// TIA Portal V18 program export: 1 tag tables, 60 data types, 57 data blocks, 79 code blocks (in call order from the OBs), 25 instance data blocks

VAR_GLOBAL   // PLC tag table "Default tag table"
   "AI11.02.01" AT %IW96 : Int;
   "AI12.01.01" AT %IW68 : Int;
   "AI12.01.02" AT %IW70 : Int;
   "AI12.01.03" AT %IW72 : Int;
   "AI12.01.04" AT %IW74 : Int;
   "AI12.01.05" AT %IW76 : Int;
   "AI12.01.06" AT %IW78 : Int;
   "AI12.01.07" AT %IW80 : Int;
   "AI12.01.08" AT %IW82 : Int;
   "AI11.02.02" AT %IW98 : Int;
   "AI11.02.03" AT %IW100 : Int;
   "AI11.02.04" AT %IW102 : Int;
   "AI11.02.05" AT %IW104 : Int;
   "AI11.02.06" AT %IW106 : Int;
   "AI11.02.07" AT %IW108 : Int;
   "AI11.02.08" AT %IW110 : Int;
   "AI11.03.01" AT %IW112 : Int;
   "AI11.03.02" AT %IW114 : Int;
   "AI11.03.03" AT %IW116 : Int;
   "AI11.03.04" AT %IW118 : Int;
   "AI11.03.05" AT %IW120 : Int;
   "AI11.03.06" AT %IW122 : Int;
   "AI11.03.07" AT %IW124 : Int;
   "AI11.03.08" AT %IW126 : Int;
   "AO12.02.01" AT %QW68 : Int;
   "AO12.02.02" AT %QW70 : Int;
   "AO12.02.03" AT %QW72 : Int;
   "AO12.02.04" AT %QW74 : Int;
   "AO12.02.05" AT %QW76 : Int;
   "AO12.02.06" AT %QW78 : Int;
   "AO12.02.07" AT %QW80 : Int;
   "AO12.02.08" AT %QW82 : Int;
   "DI12.03.01" AT %I2.0 : Bool;
   "DI12.03.02" AT %I2.1 : Bool;
   "DI12.03.03" AT %I2.2 : Bool;
   "DI12.03.04" AT %I2.3 : Bool;
   "DI12.03.05" AT %I2.4 : Bool;
   "DI12.03.06" AT %I2.5 : Bool;
   "DI12.03.07" AT %I2.6 : Bool;
   "DI12.03.08" AT %I2.7 : Bool;
   "DI12.03.09" AT %I3.0 : Bool;
   "DI12.03.10" AT %I3.1 : Bool;
   "DI12.03.11" AT %I3.2 : Bool;
   "DI12.03.12" AT %I3.3 : Bool;
   "DI12.03.13" AT %I3.4 : Bool;
   "DI12.03.14" AT %I3.5 : Bool;
   "DI12.03.15" AT %I3.6 : Bool;
   "DI12.03.16" AT %I3.7 : Bool;
   "DI12.03.17" AT %I4.0 : Bool;
   "DI12.03.18" AT %I4.1 : Bool;
   "DI12.03.19" AT %I4.2 : Bool;
   "DI12.03.20" AT %I4.3 : Bool;
   "DI12.03.21" AT %I4.4 : Bool;
   "DI12.03.22" AT %I4.5 : Bool;
   "DI12.03.23" AT %I4.6 : Bool;
   "DI12.03.24" AT %I4.7 : Bool;
   "DI12.03.25" AT %I5.0 : Bool;
   "DI12.03.26" AT %I5.1 : Bool;
   "DI12.03.27" AT %I5.2 : Bool;
   "DI12.03.28" AT %I5.3 : Bool;
   "DI12.03.29" AT %I5.4 : Bool;
   "DI12.03.30" AT %I5.5 : Bool;
   "DI12.03.31" AT %I5.6 : Bool;
   "DI12.03.32" AT %I5.7 : Bool;
   "DO12.04.01" AT %Q2.0 : Bool;
   "DO12.04.02" AT %Q2.1 : Bool;
   "DO12.04.03" AT %Q2.2 : Bool;
   "DO12.04.04" AT %Q2.3 : Bool;
   "DO12.04.05" AT %Q2.4 : Bool;
   "DO12.04.06" AT %Q2.5 : Bool;
   "DO12.04.07" AT %Q2.6 : Bool;
   "DO12.04.08" AT %Q2.7 : Bool;
   "DO12.04.09" AT %Q3.0 : Bool;
   "DO12.04.10" AT %Q3.1 : Bool;
   "DO12.04.11" AT %Q3.2 : Bool;
   "DO12.04.12" AT %Q3.3 : Bool;
   "DO12.04.13" AT %Q3.4 : Bool;
   "DO12.04.14" AT %Q3.5 : Bool;
   "DO12.04.15" AT %Q3.6 : Bool;
   "DO12.04.16" AT %Q3.7 : Bool;
   "DO12.04.17" AT %Q4.0 : Bool;
   "DO12.04.18" AT %Q4.1 : Bool;
   "DO12.04.19" AT %Q4.2 : Bool;
   "DO12.04.20" AT %Q4.3 : Bool;
   "DO12.04.21" AT %Q4.4 : Bool;
   "DO12.04.22" AT %Q4.5 : Bool;
   "DO12.04.23" AT %Q4.6 : Bool;
   "DO12.04.24" AT %Q4.7 : Bool;
   "DO12.04.25" AT %Q5.0 : Bool;
   "DO12.04.26" AT %Q5.1 : Bool;
   "DO12.04.27" AT %Q5.2 : Bool;
   "DO12.04.28" AT %Q5.3 : Bool;
   "DO12.04.29" AT %Q5.4 : Bool;
   "DO12.04.30" AT %Q5.5 : Bool;
   "DO12.04.31" AT %Q5.6 : Bool;
   "DO12.04.32" AT %Q5.7 : Bool;
   "DI11.05.01" AT %I16.0 : Bool;
   "DI11.05.02" AT %I16.1 : Bool;
   "DI11.05.03" AT %I16.2 : Bool;
   "DI11.05.04" AT %I16.3 : Bool;
   "DI11.05.05" AT %I16.4 : Bool;
   "DI11.05.06" AT %I16.5 : Bool;
   "DI11.05.07" AT %I16.6 : Bool;
   "DI11.05.08" AT %I16.7 : Bool;
   "DI11.05.09" AT %I17.0 : Bool;
   "DI11.05.10" AT %I17.1 : Bool;
   "DI11.05.11" AT %I17.2 : Bool;
   "DI11.05.12" AT %I17.3 : Bool;
   "DI11.05.13" AT %I17.4 : Bool;
   "DI11.05.14" AT %I17.5 : Bool;
   "DI11.05.15" AT %I17.6 : Bool;
   "DI11.05.16" AT %I17.7 : Bool;
   "DI11.06.01" AT %I20.0 : Bool;
   "DI11.06.02" AT %I20.1 : Bool;
   "DI11.06.03" AT %I20.2 : Bool;
   "DI11.06.04" AT %I20.3 : Bool;
   "DI11.06.05" AT %I20.4 : Bool;
   "DI11.06.06" AT %I20.5 : Bool;
   "DI11.06.07" AT %I20.6 : Bool;
   "DI11.06.08" AT %I20.7 : Bool;
   "DI11.06.09" AT %I21.0 : Bool;
   "DI11.06.10" AT %I21.1 : Bool;
   "DI11.06.11" AT %I21.2 : Bool;
   "DI11.06.12" AT %I21.3 : Bool;
   "DI11.06.13" AT %I21.4 : Bool;
   "DI11.06.14" AT %I21.5 : Bool;
   "DI11.06.15" AT %I21.6 : Bool;
   "DI11.06.16" AT %I21.7 : Bool;
   "DI11.07.01" AT %I28.0 : Bool;
   "DI11.07.02" AT %I28.1 : Bool;
   "DI11.07.03" AT %I28.2 : Bool;
   "DI11.07.04" AT %I28.3 : Bool;
   "DI11.07.05" AT %I28.4 : Bool;
   "DI11.07.06" AT %I28.5 : Bool;
   "DI11.07.07" AT %I28.6 : Bool;
   "DI11.07.08" AT %I28.7 : Bool;
   "DI11.07.09" AT %I29.0 : Bool;
   "DI11.07.10" AT %I29.1 : Bool;
   "DI11.07.11" AT %I29.2 : Bool;
   "DI11.07.12" AT %I29.3 : Bool;
   "DI11.07.13" AT %I29.4 : Bool;
   "DI11.07.14" AT %I29.5 : Bool;
   "DI11.07.15" AT %I29.6 : Bool;
   "DI11.07.16" AT %I29.7 : Bool;
   "DO11.07.01" AT %Q28.0 : Bool;
   "DO11.07.02" AT %Q28.1 : Bool;
   "DO11.07.03" AT %Q28.2 : Bool;
   "DO11.07.04" AT %Q28.3 : Bool;
   "DO11.07.05" AT %Q28.4 : Bool;
   "DO11.07.06" AT %Q28.5 : Bool;
   "DO11.07.07" AT %Q28.6 : Bool;
   "DO11.07.08" AT %Q28.7 : Bool;
   "DO11.07.09" AT %Q29.0 : Bool;
   "DO11.07.10" AT %Q29.1 : Bool;
   "DI11.08.01" AT %I32.0 : Bool;
   "DI11.08.02" AT %I32.1 : Bool;
   "DI11.08.03" AT %I32.2 : Bool;
   "DI11.08.04" AT %I32.3 : Bool;
   "DI11.08.05" AT %I32.4 : Bool;
   "DI11.08.06" AT %I32.5 : Bool;
   "DI11.08.07" AT %I32.6 : Bool;
   "DI11.08.08" AT %I32.7 : Bool;
   "DI11.08.09" AT %I33.0 : Bool;
   "DI11.08.10" AT %I33.1 : Bool;
   "DI11.08.11" AT %I33.2 : Bool;
   "DI11.08.12" AT %I33.3 : Bool;
   "DI11.08.13" AT %I33.4 : Bool;
   "DI11.08.14" AT %I33.5 : Bool;
   "DI11.08.15" AT %I33.6 : Bool;
   "DI11.08.16" AT %I33.7 : Bool;
   "DI11.01.01" AT %I0.0 : Bool;
   "DI11.01.02" AT %I0.1 : Bool;
   "DI11.01.03" AT %I0.2 : Bool;
   "DI11.01.04" AT %I0.3 : Bool;
   "DI11.01.05" AT %I0.4 : Bool;
   "DI11.01.06" AT %I0.5 : Bool;
   "DI11.01.07" AT %I0.6 : Bool;
   "DI11.01.08" AT %I0.7 : Bool;
   "DI11.01.09" AT %I1.0 : Bool;
   "DI11.01.10" AT %I1.1 : Bool;
   "DI11.01.11" AT %I1.2 : Bool;
   "DI11.01.12" AT %I1.3 : Bool;
   "DI11.01.13" AT %I1.4 : Bool;
   "DI11.01.14" AT %I1.5 : Bool;
   "DO11.07.11" AT %Q29.2 : Bool;
   "DO11.07.12" AT %Q29.3 : Bool;
   "DO11.07.13" AT %Q29.4 : Bool;
   "DO11.07.14" AT %Q29.5 : Bool;
   "DO11.07.15" AT %Q29.6 : Bool;
   "DO11.07.16" AT %Q29.7 : Bool;
   "DO11.08.01" AT %Q32.0 : Bool;
   "DO11.08.02" AT %Q32.1 : Bool;
   "DO11.08.03" AT %Q32.2 : Bool;
   "DO11.08.04" AT %Q32.3 : Bool;
   "DO11.08.05" AT %Q32.4 : Bool;
   "DO11.08.06" AT %Q32.5 : Bool;
   "DO11.08.07" AT %Q32.6 : Bool;
   "DO11.08.08" AT %Q32.7 : Bool;
   "DO11.08.09" AT %Q33.0 : Bool;
   "DO11.08.10" AT %Q33.1 : Bool;
   "DO11.08.11" AT %Q33.2 : Bool;
   "DO11.08.12" AT %Q33.3 : Bool;
   "DO11.08.13" AT %Q33.4 : Bool;
   "DO11.08.14" AT %Q33.5 : Bool;
   "DO11.08.15" AT %Q33.6 : Bool;
   "DO11.08.16" AT %Q33.7 : Bool;
   "AO11.04.01" AT %QW128 : Int;
   "AO11.04.02" AT %QW130 : Int;
   "AO11.04.03" AT %QW132 : Int;
   "AO11.04.04" AT %QW134 : Int;
   "DO11.01.01" AT %Q0.0 : Bool;
   "DO11.01.02" AT %Q0.1 : Bool;
   "DO11.01.03" AT %Q0.2 : Bool;
   "DO11.01.04" AT %Q0.3 : Bool;
   "DO11.01.05" AT %Q0.4 : Bool;
   "DO11.01.06" AT %Q0.5 : Bool;
   "DO11.01.07" AT %Q0.6 : Bool;
   "DO11.01.08" AT %Q0.7 : Bool;
   "DO11.01.09" AT %Q1.0 : Bool;
   "DO11.01.10" AT %Q1.1 : Bool;
   "AI11.01.01" AT %IW64 : Int;
   "AI11.01.02" AT %IW66 : Int;
   "AO11.01.01" AT %QW64 : Int;
   "AO11.01.02" AT %QW66 : Int;
   System_Byte AT %MB1 : Byte;
   FirstScan AT %M1.0 : Bool;
   DiagStatusUpdate AT %M1.1 : Bool;
   AlwaysTRUE AT %M1.2 : Bool;
   AlwaysFALSE AT %M1.3 : Bool;
   Clock_Byte AT %MB0 : Byte;
   Clock_10Hz AT %M0.0 : Bool;
   Clock_5Hz AT %M0.1 : Bool;
   "Clock_2.5Hz" AT %M0.2 : Bool;
   Clock_2Hz AT %M0.3 : Bool;
   "Clock_1.25Hz" AT %M0.4 : Bool;
   Clock_1Hz AT %M0.5 : Bool;
   "Clock_0.625Hz" AT %M0.6 : Bool;
   "Clock_0.5Hz" AT %M0.7 : Bool;
   Lux AT %MD20 : Real;
   "DI12.05.01" AT %I6.0 : Bool;
   "DI12.05.02" AT %I6.1 : Bool;
   "DI12.05.03" AT %I6.2 : Bool;
   "DI12.05.04" AT %I6.3 : Bool;
   "DI12.05.05" AT %I6.4 : Bool;
   "DI12.05.06" AT %I6.5 : Bool;
   "DI12.05.07" AT %I6.6 : Bool;
   "DI12.05.08" AT %I6.7 : Bool;
   "DI12.05.09" AT %I7.0 : Bool;
   "DI12.05.10" AT %I7.1 : Bool;
   "DI12.05.11" AT %I7.2 : Bool;
   "DI12.05.12" AT %I7.3 : Bool;
   "DI12.05.13" AT %I7.4 : Bool;
   "DI12.05.14" AT %I7.5 : Bool;
   "DI12.05.15" AT %I7.6 : Bool;
   "DI12.05.16" AT %I7.7 : Bool;
   OAT_clock_triger AT %M5.0 : Bool;
   "Run/Stop" AT %M5.1 : Bool;
   rAO_temporary AT %MD60 : Real;
   rAI_temporary AT %MD61 : Real;
   xDO_temporary AT %M5.2 : Bool;   //    {ExternalWritable false}
   xDI_temporary AT %M5.3 : Bool;
   iUnitStateCounter AT %MW66 : Int;
   iTargetUnitStareCounter AT %MW68 : Int;
   cTargetUnitStatePrevOne AT %MB8 : Byte;
   cActualOpModePrevOne AT %MB9 : Byte;
   iActualOpModeCounter AT %MW10 : Int;
   xDL_Pump1_Run AT %M12.0 : Bool;
   xDL_Pump2_Run AT %M12.1 : Bool;
END_VAR
VAR_GLOBAL CONSTANT   // user constants
   IOmark_string_length : Int := 25;
   DIbasic_OnDelayCycle : Int := 800;
   DIbasic_OffDelayCycle : Int := 800;
END_VAR

TYPE "UDT_DailyScheduler"
// stored: IsFailsafeCompliant false
   STRUCT
      Start : Time_Of_Day;
      Stop : Time_Of_Day;
   END_STRUCT;
END_TYPE

TYPE "UDT_Store_OpMode"
// stored: IsFailsafeCompliant false
   STRUCT
      cPreviousOne { S7_SetPoint := 'True'} : Byte;
      cActual { S7_SetPoint := 'True'} : Byte;   // Поточний/Актуальний режим роботи
      cTarget { S7_SetPoint := 'True'} : Byte;   // Вибраний режим роботи, але ще не дійшли до нього
      cPreselectedOpMode : Byte;   // 0-Protection/1-economy/2-PreComfort/3-Comfort/4-Auto
   END_STRUCT;
END_TYPE

TYPE "UDT_Store_Setpoints"
// stored: IsFailsafeCompliant false
   STRUCT
      Room : Struct
         Actual : Struct
            rRATHeating : Real;
            rRATCooling : Real;
            rIAQ : Real;
            rBuildingdP : Real;
         END_STRUCT;
         Comfort : Struct
            rRATHeating : Real := 18.0;
            rRATCooling : Real := 22.0;
            rIAQ : Real := 600.0;
            rBuildingdP : Real := 5.0;
         END_STRUCT;
         PreComfort : Struct
            rRATHeating : Real := 16.0;
            rRATCooling : Real := 25.0;
            rIAQ : Real := 800.0;
            rBuildingdP : Real := 2.0;
         END_STRUCT;
         Econom : Struct
            rRATHeating : Real := 15.0;
            rRATCooling : Real := 30.0;
            rIAQ : Real;
            rBuildingdP : Real;
         END_STRUCT;
         Protection : Struct
            rRATHeating : Real := 5.0;
            rRATCooling : Real := 35.0;
            rIAQ : Real := 0.0;
            rBuildingdP : Real := 0.0;
         END_STRUCT;
      END_STRUCT;
   END_STRUCT;
END_TYPE

TYPE "UDT_WeatherCompCurve"
// stored: IsFailsafeCompliant false
   STRUCT
      rEffectiveRoomSetPoint : Array[0..2] of Real;
      rHeatingCurveLevel : Array[0..2] of Real;
      rHeatingCurveSlope : Array[0..2] of Real;
      rSetpointTemp : Array[0..2] of Real;
      rOATforHeatingCurves : Array[0..2] of Real;
   END_STRUCT;
   // rEffectiveRoomSetPoint[0] := 20.0;
   // rEffectiveRoomSetPoint[1] := 21.0;
   // rEffectiveRoomSetPoint[2] := 22.0;
   // rHeatingCurveLevel[1] := 1.0;
   // rHeatingCurveLevel[2] := 2.0;
   // rHeatingCurveSlope[0] := 2.0;
   // rHeatingCurveSlope[1] := 2.1;
   // rHeatingCurveSlope[2] := 2.2;
   // rSetpointTemp[0] := 50.0;
   // rSetpointTemp[1] := 51.0;
   // rSetpointTemp[2] := 52.0;
END_TYPE

TYPE "UDT_OAT"
// stored: IsFailsafeCompliant false
   STRUCT
      rOAT_PLC_IO : Real;
      rOAT_WeatherStation : Real;
      rOAT_Boilers : Real;
      rOAT_Actual : Real;
   END_STRUCT;
END_TYPE

TYPE "UDT_Store_Holidays"
// stored: IsFailsafeCompliant false
   STRUCT
      UDT_Store_Holidays : Array[0..7] of Date;
   END_STRUCT;
END_TYPE

TYPE "UDT_Store_Scheduler"
// stored: IsFailsafeCompliant false
   STRUCT
      cOpModeNowByScheduler : Byte;
      Monday : Struct
         Comfort { S7_SetPoint := 'True'} : "UDT_DailyScheduler";
         PreComfort { S7_SetPoint := 'True'} : "UDT_DailyScheduler";
      END_STRUCT;
      WorkingDays : Struct
         Comfort { S7_SetPoint := 'True'} : "UDT_DailyScheduler";
         PreComfort { S7_SetPoint := 'True'} : "UDT_DailyScheduler";
      END_STRUCT;
      Saturday : Struct
         Comfort { S7_SetPoint := 'True'} : "UDT_DailyScheduler";
         PreComfort { S7_SetPoint := 'True'} : "UDT_DailyScheduler";
      END_STRUCT;
      Sunday : Struct
         Comfort { S7_SetPoint := 'True'} : "UDT_DailyScheduler";
         PreComfort { S7_SetPoint := 'True'} : "UDT_DailyScheduler";
      END_STRUCT;
      Holiday : Struct
         Comfort { S7_SetPoint := 'True'} : "UDT_DailyScheduler";
         PreComfort { S7_SetPoint := 'True'} : "UDT_DailyScheduler";
      END_STRUCT;
   END_STRUCT;
END_TYPE

TYPE "UDT_Store_Season"
// stored: IsFailsafeCompliant false
   STRUCT
      cSeasonModeSelection : Byte;   // 0 = Summer 1 = Winter 2 = Midseason, 3=Auro
      cActual : Byte;   // 0 = Summer 1 = Winter 2 = Midseason
      cTarget : Byte;
      cReserve : Byte;
      rOATtoWinter : Real := 10.0;
      rOATtoSummer : Real := 12.0;
   END_STRUCT;
END_TYPE

TYPE "UDT_DL_Vars"
// stored: IsFailsafeCompliant false
   STRUCT
      rOATtoHeatUpLine : Real;
      cReserve1 : Byte;
      cReserve2 : Byte;
      cDLPanelModeSelector : Byte := 16#3;
      rDayTankLevelAlarmMin : Array[1..2] of Real;
      rDayTankLevelStartFilling : Array[1..2] of Real;
      rDayTankLevelStopFilling : Array[1..2] of Real;
      rDayTankLevelAlarmMax : Array[1..2] of Real;
      cExericeSeconds : Array[1..2] of Byte;
      cMaxHoursWithoutRunToExerise : Array[1..2] of Byte;
      cActualHoursWithoutRunToExerise : Array[1..2] of Byte;
   END_STRUCT;
   // rDayTankLevelAlarmMin[1] := 50.0;
   // rDayTankLevelAlarmMin[2] := 51.0;
   // rDayTankLevelStartFilling[1] := 70.0;
   // rDayTankLevelStartFilling[2] := 71.0;
   // rDayTankLevelStopFilling[1] := 90.0;
   // rDayTankLevelStopFilling[2] := 91.1;
   // rDayTankLevelAlarmMax[1] := 95.0;
   // rDayTankLevelAlarmMax[2] := 96.0;
   // cExericeSeconds[1..2] := 16#FA;
   // cMaxHoursWithoutRunToExerise[1] := 16#A8;
   // cMaxHoursWithoutRunToExerise[2] := 16#A9;
END_TYPE

TYPE "UDT_BoilersOnOffSettings"
// stored: IsFailsafeCompliant false
   STRUCT
      OAT : Struct
         rBoiler1OATOff : Real := 18.0;
         rBoiler1OATOn : Real := 15.0;
         rBoiler2OAT1On : Real := 5.0;
         rBoiler2OAT1Off : Real := 10.0;
         rBoiler2OAT2On : Real := -5.0;
         rBoiler2OAT2Off : Real;
      END_STRUCT;
      PLCModeSelection : Struct
         cPreselectedOpModePLC : Byte;   // Вибор режиму роботи з PLC. 0-Вимкенено/1-Boiler1/2-Boiler2/3-B1+B2/4-Auto
         cActualOpModePLC : Byte;   // Актуальний режим роботи з PLC. 0-Вимкенено/1-Boiler1/2-Boiler2/3-B1+B2/4-Auto
      END_STRUCT;
   END_STRUCT;
END_TYPE

TYPE "UDT_Vitotronic100_Alarms"
// stored: IsFailsafeCompliant false
   STRUCT
      "00 General alarm" : Array[0..2] of Bool;
   END_STRUCT;
END_TYPE

TYPE "UDT_Vitotronic100_IOs"
// stored: IsFailsafeCompliant false
   STRUCT
      "Boiler water temperature" : Array[0..2] of Real;
      "Flue gas temperature" : Array[0..2] of Real;
      "Return temperature 17A" : Array[0..2] of Real;
      "Return temperature 17B" : Array[0..2] of Real;
   END_STRUCT;
END_TYPE

TYPE "UDT_Vitotronic100_Params"
// stored: IsFailsafeCompliant false
   STRUCT
      "Actual system output - value" : Array[0..2] of Real;
      "Boiler output value" : Array[0..2] of Real;
      "Burner output" : Array[0..2] of Real;
      "Maximum boiler temperature" : Array[0..2] of Real;
      "Minimum boiler temperature" : Array[0..2] of Real;
      "Set boiler output (effective)" : Array[0..2] of Real;
      "Set boiler water temperature (effective)" : Array[0..2] of Real;
   END_STRUCT;
END_TYPE

TYPE "UDT_BoilersSummaryAlarms"
// stored: IsFailsafeCompliant false
   STRUCT
      BlockingAlarm : Array[1..2] of Bool;
   END_STRUCT;
END_TYPE

TYPE "UDT_Vitotronic100_Settings"
// stored: IsFailsafeCompliant false
   STRUCT
      "Set boiler water temperature" : Array[0..2] of Real;
      "Operating mode system_boiler" : Array[0..2] of Int;
   END_STRUCT;
END_TYPE

TYPE "UDT_BoilerOpMode"
// stored: IsFailsafeCompliant false
   STRUCT
      cPreviousOne { S7_SetPoint := 'True'} : Array[1..2] of Byte;
      cActual { S7_SetPoint := 'True'} : Array[1..2] of Byte;   // Поточний/Актуальний режим роботи
      cTarget { S7_SetPoint := 'True'} : Array[1..2] of Byte;   // Вибраний режим роботи, але ще не дійшли до нього
      cPreselectedOpModePLC : Array[1..2] of Byte;   // Вибор режиму роботи з PLC. 0-Вимкенено/1-Boiler1/2-Boiler2/3-B1+B2/4-Auto
      cReserve : Array[1..2] of Byte;
      cPreselectedOpModePanel : Array[1..2] of Byte;   // Вибор режиму роботи з Фізичного перемикача на шафы. 0-Summer/1-Winter/2--Auto
      xBoiler2IndividualPanelSwitch : Bool;
   END_STRUCT;
END_TYPE

TYPE "UDT_BoilerUnitState"
// stored: IsFailsafeCompliant false
   STRUCT
      iBoilerSimpleState : Array[1..2] of Int;   // 0-Off, 1 - Heating, 2 - Alarm
      xBoilerOATRequest : Array[1..2] of Bool;
      xBoilerRequestedByAlarm : Array[1..2] of Bool;
      cTarget : Array[1..2] of Byte;
      cActual : Array[1..2] of Byte;
   END_STRUCT;
END_TYPE

TYPE "UDT_AIbasic"
// stored: IsFailsafeCompliant false
   STRUCT
      iID : DInt;   // AIs ID for monitoring
      iValue : Int;   // Int value
      rValue : Real;   // Real value
      iFilterSet : Int;   // Filter value
      rMin : Real;   // Scale Min
      rMax : Real;   // Scale Max
      wMark : String["IOmark_string_length"];   // AIs label for monitoring
   END_STRUCT;
END_TYPE

TYPE "UDT_AObasic"
// stored: IsFailsafeCompliant false
   STRUCT
      iID : DInt;   // AOs ID for monitoring
      rInput : Real;   // Value for AO
      cMOA : Byte;   // Mode Manual/Off/Auto
      rMan_output : Real;   // Manual output
      iOutput : Int;   // Output for DAC
      wMark : String["IOmark_string_length"];   // AOs label for monitoring
   END_STRUCT;
END_TYPE

TYPE "UDT_DIbasic"
// stored: IsFailsafeCompliant false
   STRUCT
      iID : DInt;   // DIs ID for monitoring
      iCounter : Int;   // Counter for DIs EDGE
      xFiltered : Bool;   // Filtered value
      wMark : String["IOmark_string_length"];   // DIs label for monitoring
      iAddImpOff : Int;   // Temp
      iAddImpOn : Int;   // Temp
      xMemory : Bool;   // Temp
   END_STRUCT;
END_TYPE

TYPE "UDT_DObasic"
// stored: IsFailsafeCompliant false
   STRUCT
      iID : DInt;   // DOs ID for monitoring
      xInput : Bool;   // Value for DO
      cMOA : Byte;   // Mode Manual/Off/Auto
      xOutput : Bool;   // Phisicl output
      iCounter : Int;   // Counter
      Mark : String["IOmark_string_length"];   // DOs label for monitoring
      xBitCount : Bool;   // Internal
   END_STRUCT;
END_TYPE

TYPE "UDT_RTDbasic"
// stored: IsFailsafeCompliant false
   STRUCT
      iID : DInt;   // AIs ID for monitoring
      rValue : Real;   // Real value
      iFilterSet : Int;   // Filter value
      rCalibration : Real;   // Scale Min
      rDiv : Real := 100.0;   // Scale Max
      wMark : String["IOmark_string_length"];   // AIs label for monitoring
   END_STRUCT;
END_TYPE

TYPE "UDT_DLsAI"
// stored: IsFailsafeCompliant false
   STRUCT
      rDayTankLevel : Array[1..2] of Real;   // 10.82(3) Рівень палива в баку добового запасу ДГУ1(2)
   END_STRUCT;
END_TYPE

TYPE "UDT_DLsDI"
// stored: IsFailsafeCompliant false
   STRUCT
      xDieselLineHeatingReady : Array[1..2] of Bool;
      xDieselLineHeatingInd : Array[1..2] of Bool;
      xDieselLinePumpInd : Array[1..2] of Bool;
      xDieselLinePnom : Bool;   // 10.67 Номінальний тиск в ДП ліній
      xDieselLineValveToBoilerInd : Bool;   // 10.66 Клапанна група на Котел
      xDieselLinePmax : Bool;   // 10.68 Високий тиск в ДП ліній
      xDieselLinePumpZoneWaterFloodAlarm : Bool;   // 10.79 Затоплення приямку з насосами
      xDieselLineMainTankDoubleWallAlarmInd : Bool;   // 10.63 62 SGB DL-4000
      xDieselLineMainTankMinLevelInd : Bool;   // 10.75 76
      Reserve1 : Bool;
      Reserve2 : Bool;
      xDieselLinePumpPanelSelectorOff : Bool;
      xDieselLinePumpPanelSelectorP1Man : Bool;
      xDieselLinePumpPanelSelectorP2Man : Bool;
      xDieselLinePumpPanelSelectorAuto : Bool;
   END_STRUCT;
END_TYPE

TYPE "UDT_DLsDO"
// stored: IsFailsafeCompliant false
   STRUCT
      xDieselLineHeatingCmd : Array[1..2] of Bool;
      xDieselLinePumpEnable : Bool;
      xDieselLinePumpSelect : Bool;
      xDieselLineDayTankValve : Array[1..2] of Bool;
      Reserve : Array[1..2] of Bool;
   END_STRUCT;
END_TYPE

TYPE "AHUChannel_v1"
// stored: IsFailsafeCompliant false
   STRUCT
      SAFCmd1 : Array[0..2] of Bool;
      SAFCmd2 : Array[0..2] of Bool;
      SAFCmd3 : Array[0..2] of Bool;
      SAFSpeed1Ind : Array[0..2] of Bool;   // Off/On
      SAFSpeed2Ind : Array[0..2] of Bool;   // Off/On
      SAFIsBlockedByFrostProt : Array[0..2] of Bool;   // Off/On
      SAFInd4 : Array[0..2] of Bool;
      SAFInd5 : Array[0..2] of Bool;
      SAFInd6 : Array[0..2] of Bool;
      SAFInd7 : Array[0..2] of Bool;
      HeaterRlyIsOn : Array[0..2] of Bool;   // Off/On
      HeaterRlyIsOff : Array[0..2] of Bool;   // Off/On
      HeaterRlyOnCmd : Array[0..2] of Bool;   // Off/On
      HeaterInitialSignal : Array[0..2] of Real;   // 0-100.0%
      HeaterAdaptedSignal : Array[0..2] of Real;   // 0-100.0%
      MixingRlyIsOn : Array[0..2] of Bool;   // Off/On
      MixingRlyIsOff : Array[0..2] of Bool;   // Off/On
      MixingRlyOnCmd : Array[0..2] of Bool;   // Off/On
      MixingInitialSignal : Array[0..2] of Real;   // 0-100.0%
      MixingAdaptedSignal : Array[0..2] of Real;   // 0-100.0%
      ExtractRlyIsOn : Array[0..2] of Bool;   // Off/On
      ExtractRlyIsOff : Array[0..2] of Bool;   // Off/On
      ExtractRlyOnCmd : Array[0..2] of Bool;   // Off/On
      ExtractInitialSignal : Array[0..2] of Real;   // 0-100.0%
      ExtractAdaptedSignal : Array[0..2] of Real;   // 0-100.0%
   END_STRUCT;
END_TYPE

TYPE "SupplyFanChannel_v1"
// stored: IsFailsafeCompliant false
   STRUCT
      SAFSpeed1Ind : Array[0..2] of Bool;   // Off/On
      SAFSpeed2Ind : Array[0..2] of Bool;   // Off/On
      SAFIsBlockedByFrostProt : Array[0..2] of Bool;   // Off/On
   END_STRUCT;
END_TYPE

TYPE "AnalogChannel_v0"
// stored: IsFailsafeCompliant false
   STRUCT
      CHRlyIsOn : Array[0..11] of Bool;   // Off/On
      CHRlyIsOff : Array[0..11] of Bool;   // Off/On
      CHRlyOnCmd : Array[0..11] of Bool;   // Off/On
      CHInitialSignal : Array[0..11] of Real;   // 0-100.0%
      CHAdaptedSignal : Array[0..11] of Real;   // 0-100.0%
   END_STRUCT;
END_TYPE

TYPE "UDT_AnalogProxyCH_Vars"
// stored: IsFailsafeCompliant false
   STRUCT
      cCHModeCtrl : Array[1..8] of Byte;   // 0-Not Active, 1-StraigntSignal,2-Adapt , 3-NewSignal
      xCHRlyIsOnInd : Array[1..8] of Bool;   // Off/On
      xCHRlyIsOffInd : Array[1..8] of Bool;   // Off/On
      xCHRlyOnCmd : Array[1..8] of Bool;   // Off/On
      xCHRlyIndError : Array[1..8] of Bool;   // Norm/Alarm
      rCHDrivenSignal : Array[1..8] of Real;   // 0-100.0%
      rCHProxySignal : Array[1..8] of Real;   // 0-100.0%
   END_STRUCT;
END_TYPE

TYPE "UDT_AHUSummaryAlarms"
// stored: IsFailsafeCompliant false
   STRUCT
      FrostAlarm : Array[1..3] of Bool;   // 0Active/Uack 0 - no blocking alarms/ 1- blocking alarms/ 2- frost alrm
      BlockingAlarm : Array[1..3] of Bool;
      HeaterPump : Array[1..3] of Bool;
      SAFAlarm : Array[1..3] of Bool;
      SAFilterAlarm : Array[1..3] of Bool;
   END_STRUCT;
END_TYPE

TYPE "UDT_AHUEqpDataType"
// stored: IsFailsafeCompliant false
   STRUCT
      cFan : Array[1..3] of Byte;   // 0-wout ctrl/1 - ProxiAdaptation/
      cExtractDumper : Array[1..3] of Byte;   // 0-wout ctrl/1 - ProxiAdaptation/
      cMixingDumper : Array[1..3] of Byte;   // 0-wout ctrl/1 - ProxiAdaptation/
      cHeater : Array[1..3] of Byte;   // 0-wout ctrl/1 - ProxiAdaptation/
      cCooler : Array[1..3] of Byte;   // 0-wout ctrl/1 - ProxiAdaptation/
      cWHU : Array[1..3] of Byte;   // 0-wout ctrl/1 - ProxiAdaptation/
   END_STRUCT;
END_TYPE

TYPE "UDT_AHUEqpDemand"
// stored: IsFailsafeCompliant false
   STRUCT
      rFan : Array[1..3] of Real;   // 0-wout ctrl/1 - ProxiAdaptation/
      rExtractDumper : Array[1..3] of Real;   // 0-wout ctrl/1 - ProxiAdaptation/
      rMixingDumper : Array[1..3] of Real;   // 0-wout ctrl/1 - ProxiAdaptation/
      rHeater : Array[1..3] of Real;   // 0-wout ctrl/1 - ProxiAdaptation/
      rCooler : Array[1..3] of Real;   // 0-wout ctrl/1 - ProxiAdaptation/
      rWHU : Array[1..3] of Real;   // 0-wout ctrl/1 - ProxiAdaptation/
   END_STRUCT;
END_TYPE

TYPE "UDT_AHUsAI"
// stored: IsFailsafeCompliant false
   STRUCT
      rIAQ : Array[1..3] of Real;   // Рівень концентрації СО2 в торговій залі, ppm
      rBuildingdP : Array[1..3] of Real;   // Перепад тиску між будівлею і вулицею, Pa
      rRoomAirTemp_PLC_AI : Array[1..3] of Real;   // Температура повітря в торговій залі з вх PLC, C
      rSupplyAirTemp : Array[1..3] of Real;   // Температура повітря що подається з AHU в торгову залу, C
      rReturnAirTemp : Array[1..3] of Real;   // Температура повітря що подається з торгової зали в AHU, C
      rFrostProtWaterTemp : Array[1..3] of Real;   // Температура зворотнього теплоносія, C
      rFrostProtAirTemp : Array[1..3] of Real;   // Температура повытря пысля ТО, C x.50
      rRoomAirRelHumi : Array[1..3] of Real;
      rReserve : Array[1..3] of Real;   // Вулична температура x.99, C
      rSAFilterdP : Array[1..3] of Real;   // Перепад тиску на приточному filter x.53
      rSAFFlow : Array[1..3] of Real;   // Витрата повытря на припливному вентиляторы
      rRoomAirTemp_Actual : Array[1..3] of Real;   // Температура повітря в торговій залі Вираховане, C
      rRoomAirTemp_LoraAvg : Array[1..3] of Real;   // Температура повітря в торговій залі Вираховане, C
      rRoomAirTemp_MSensor : Array[1..3] of Real;   // Температура повітря в торговій залі Вираховане, C
      rReserve_1 : Array[1..3] of Real;
      rReserve_2 : Array[1..3] of Real;
      rReserve_3 : Array[1..3] of Real;
      rReserve_4 : Array[1..3] of Real;
      rReserve_5 : Array[1..3] of Real;
      rReserve_6 : Array[1..3] of Real;
      rReserve_7 : Array[1..3] of Real;
      rReserve_8 : Array[1..3] of Real;
      rReserve_9 : Array[1..3] of Real;
      cRoomTempSelect : Array[1..3] of Byte;   // 0=PLC_IO, 1=LoraAvg, 2=MSensor,3 =Auto
   END_STRUCT;
   // cRoomTempSelect[1] := 1;
   // cRoomTempSelect[2] := 0;
END_TYPE

TYPE "UDT_AHUsDI"
// stored: IsFailsafeCompliant false
   STRUCT
      xHeaterPumpReady : Array[1..3] of Bool;
      xHeaterPumpInd : Array[1..3] of Bool;
      xHeaterPumpAlarm : Array[1..3] of Bool;
      xSAFAnalogReady : Array[1..3] of Bool;
      xSAFAnalogInd : Array[1..3] of Bool;
      xSAFAnalogAlarm : Array[1..3] of Bool;
      xSAFSp1Ready : Array[1..3] of Bool;
      xSAFSp1Ind : Array[1..3] of Bool;
      xSAFSp1Alarm : Array[1..3] of Bool;
      xSAFSp2Ready : Array[1..3] of Bool;
      xSAFSp2Ind : Array[1..3] of Bool;
      xSAFSp2Alarm : Array[1..3] of Bool;
      xSAFdPInd : Array[1..3] of Bool;
      xFrostProtTstat : Array[1..3] of Bool;
      xSAFdPAlarm : Array[1..3] of Bool;
      xSAFPanelSelectorOff : Array[1..3] of Bool;
      xSAFPanelSelector1St : Array[1..3] of Bool;
      xSAFPanelSelector2St : Array[1..3] of Bool;
      xSAFPanelSelectorAuto : Array[1..3] of Bool;
      xSAFMotorPTCAlarm : Array[1..3] of Bool;
      xServiceSwitchOnAHU : Array[1..3] of Bool;
      xCoolerAlarm : Array[1..3] of Bool;
      xCoolerC1Ind : Array[1..3] of Bool;
      xCoolerC2Ind : Array[1..3] of Bool;
      xFilterdP : Array[1..3] of Bool;
      xHeaterPumpModeInAuto : Array[1..3] of Bool;
   END_STRUCT;
END_TYPE

TYPE "UDT_AHUsDO"
// stored: IsFailsafeCompliant false
   STRUCT
      xHeaterPumpCmd : Array[1..3] of Bool;
      xSAFAnalogEnable : Array[1..3] of Bool;
      xSAFSp1Cmd : Array[1..3] of Bool;
      xSAFSp2Cmd : Array[1..3] of Bool;
      xCoolerSt1Cmd : Array[1..3] of Bool;
      xCoolerSt2Cmd : Array[1..3] of Bool;
      xCoolerSt3Cmd : Array[1..3] of Bool;
      xCoolerSt4Cmd : Array[1..3] of Bool;
   END_STRUCT;
END_TYPE

TYPE "UDT_FrostProtection"
// stored: IsFailsafeCompliant false
   STRUCT
      AlarmWaterTempLimit : Array[1..3] of Real;
      BandMin : Array[1..3] of Real;
      BandMax : Array[1..3] of Real;
      OATMin : Array[1..3] of Real;
      OATMax : Array[1..3] of Real;
      CalculatedAddition : Array[1..3] of Real;
      OATtoStartPreheating : Array[1..3] of Real;
   END_STRUCT;
END_TYPE

TYPE "UTD_AHUsAO"
// stored: IsFailsafeCompliant false
   STRUCT
      rSAFAnalog : Array[1..3] of Real;
      rHeater : Array[1..3] of Real;
      rMixingAirDumper : Array[1..3] of Real;
      rExtractAirDumper : Array[1..3] of Real;
      rCooler : Array[1..3] of Real;
      rWHU : Array[1..3] of Real;
   END_STRUCT;
END_TYPE

TYPE "UDT_AHUsState"
// stored: IsFailsafeCompliant false
   STRUCT
      cPreviousOne : Array[1..3] of Byte;
      cActual : Array[1..3] of Byte;
      cTarget : Array[1..3] of Byte;
      xActualStateEdge : Array[1..3] of Bool;
      cSimpleForHMI : Array[1..3] of Byte;
      iCounterOfSwitchingBtwActualStates : Array[1..3] of Int;
   END_STRUCT;
   // // cSimpleForHMI[1] : 0 - Not Exist, 1-Stopped, 1- Run, 2 - Alarm Blocked
   // // cSimpleForHMI[2] : 0 - Not Exist, 1-Stopped, 1- Run, 2 - Alarm Blocked
   // // cSimpleForHMI[3] : 0 - Not Exist, 1-Stopped, 1- Run, 2 - Alarm Blocked
END_TYPE

TYPE "UDT_AHUsStsDelay"
// stored: IsFailsafeCompliant false
   STRUCT
      cCnt : Array[1..3] of Byte;
      cCheckingUpTime : Array[1..3] of Byte;
      cPreheatingTime : Array[1..3] of Byte;
      cStartingTime : Array[1..3] of Byte;
      cStoppingTime : Array[1..3] of Byte;
      cWorkOnFullRecycleTime : Array[1..3] of Byte;
   END_STRUCT;
   // cCheckingUpTime[1..2] := 10;
   // cPreheatingTime[1..2] := 20;
   // cStartingTime[1..2] := 10;
   // cStoppingTime[1..2] := 10;
END_TYPE

TYPE "UDT_AHUsRegDemand"
// stored: IsFailsafeCompliant false
   STRUCT
      rHeating : Array[1..3] of Real;
      rCooling : Array[1..3] of Real;
      rIAQ : Array[1..3] of Real;
      rBuildingPressure : Array[1..3] of Real;
      rFreshAirTemp : Array[1..3] of Real;
      rFrostProtection : Array[1..3] of Real;
      rFreshAirSummary : Array[1..3] of Real;
   END_STRUCT;
END_TYPE

TYPE "UDT_AHUsRegulators"
// stored: IsFailsafeCompliant false
   STRUCT
      Cfg : "UDT_AHUsRegulatorsDataType";
      State : "UDT_AHUsRegulatorsDataType";
      Demands { S7_SetPoint := 'True'} : "UDT_AHUsRegDemand";
      FreshAirCoef { S7_SetPoint := 'True'} : "UDT_AHUsFreshAirCoef";
   END_STRUCT;
END_TYPE

TYPE "UDT_AHUsSustainedRequests"
// stored: IsFailsafeCompliant false
   STRUCT
      xNightCooling : Array[1..3] of Bool;
      xSustainedOnCooling : Array[1..3] of Bool;
      xSustainedOnHeating : Array[1..3] of Bool;
      xSusteinedOnIAQ : Array[1..3] of Bool;
      xSusteainedOnBuildingdP : Array[1..3] of Bool;
      cSummarySustTempRequest : Array[1..3] of Byte;
      xStartRequest : Array[1..3] of Bool;
      xBlockRequest : Array[1..3] of Bool;
   END_STRUCT;
END_TYPE

TYPE "UDT_AHUSetpoints"
// stored: IsFailsafeCompliant false
   STRUCT
      Room : Struct
         Actual { S7_SetPoint := 'True'} : "UDT_SetPointsBasic";
         Target { S7_SetPoint := 'True'} : "UDT_SetPointsBasic";
         Shift { S7_SetPoint := 'True'} : "UDT_SetPointsBasic";
      END_STRUCT;
      Supply { S7_SetPoint := 'True'} : "UDT_AHUsSATSetPoints";
   END_STRUCT;
   // Room.Shift.RATHeating[1..2] := 0.0;
   // Room.Shift.RATCooling[1..2] := 0.0;
   // Room.Shift.IAQ[1..2] := 0.0;
   // Room.Shift.BuildingdP[1..2] := 0.0;
END_TYPE

TYPE "UDT_AHUsSATSetPoints"
// stored: IsFailsafeCompliant false
   STRUCT
      Actual { S7_SetPoint := 'True'} : Array[1..3] of Real;
      Target : Array[1..3] of Real;
      MinAbs : Array[1..3] of Real;
      MaxAbs : Array[1..3] of Real;
   END_STRUCT;
END_TYPE

TYPE "UDT_SetPointsBasic"
// stored: IsFailsafeCompliant false
   STRUCT
      RATHeating : Array[1..3] of Real;   // C
      RATCooling : Array[1..3] of Real;   // C
      IAQ : Array[1..3] of Real;   // ppm
      BuildingdP : Array[1..3] of Real;   // Pa
   END_STRUCT;
   // RATHeating[1..2] := 20.0;
   // RATCooling[1..2] := 22.0;
   // IAQ[1..2] := 800.0;
   // BuildingdP[1..2] := 5.0;
END_TYPE

TYPE "UDT_HSsAI"
// stored: IsFailsafeCompliant false
   STRUCT
      rHSBoilerRoomTemp : Real;   // 10.10 Температура в котельный
      rHSWaterPressure : Real;   // 10.09 Тиск в системы опалення
      rHSSupplyMainfoldTemp : Real;
      rOutdoorTemp_PLC_AI : Real;
   END_STRUCT;
END_TYPE

TYPE "UDT_HSsDI"
// stored: IsFailsafeCompliant false
   STRUCT
      xBoilerShuntPumpReady : Array[1..2] of Bool;
      xBoilerShuntPumpInd : Array[1..2] of Bool;
      xBoilerShuntPumpAlarm : Array[1..2] of Bool;
      xBoilerShuntPumpInAuto : Array[1..2] of Bool;
      xBoilerStage1Ind : Array[1..2] of Bool;
      xBoilerStage2Ind : Array[1..2] of Bool;
      xBurnerAlarm : Array[1..2] of Bool;
      xBoilerAlarm : Array[1..2] of Bool;
      xBoilerReady : Array[1..2] of Bool;
      xBoilerReserve : Array[1..2] of Bool;
      xSeasonWinter : Array[1..2] of Bool;
      xSeasonSummer : Array[1..2] of Bool;
      xSeasonAuto : Array[1..2] of Bool;
      xBoilerWaterLvl : Array[1..2] of Bool;
      xBoilerPmin : Array[1..2] of Bool;
      xBoilerPmax : Array[1..2] of Bool;
   END_STRUCT;
   // xBoilerShuntPumpReady[1..2] := true;
END_TYPE

TYPE "UDT_HCsDI"
// stored: IsFailsafeCompliant false
   STRUCT
      xHCPump1Ready : Array[1..2] of Bool;
      xHCPump1Ind : Array[1..2] of Bool;
      xHCPump1Alarm : Array[1..2] of Bool;
      xHCPump2Ready : Array[1..2] of Bool;
      xHCPump2Ind : Array[1..2] of Bool;
      xHCPump2Alarm : Array[1..2] of Bool;
      xHCDoublePumpInAuto : Array[1..2] of Bool;
   END_STRUCT;
   // xHCPump1Ready[1..2] := true;
   // xHCPump2Ready[1..2] := true;
END_TYPE

TYPE "UDT_HCsDO"
// stored: IsFailsafeCompliant false
   STRUCT
      xHC3wvIncrease : Array[1..2] of Bool;
      xHC3wvDecrease : Array[1..2] of Bool;
      xHCPump1Cmd : Array[1..2] of Bool;
      xHCPump2Cmd : Array[1..2] of Bool;
   END_STRUCT;
END_TYPE

TYPE "UDT_AHsDO"
// stored: IsFailsafeCompliant false
   STRUCT
      xAHCentralEnable : Bool;
   END_STRUCT;
END_TYPE

TYPE "UDT_AHUEqp"
// stored: IsFailsafeCompliant false
   STRUCT
      Cfg : "UDT_AHUEqpDataType";
      State { S7_SetPoint := 'True'} : "UDT_AHUEqpDataType";
      Demand { S7_SetPoint := 'True'} : "UDT_AHUEqpDemand";
      LimiterGridOperation { S7_SetPoint := 'True'} : "UDT_AHUsEqpDemandLimiter";
      LimiterDieselOperation { S7_SetPoint := 'True'} : "UDT_AHUsEqpDemandLimiter";
   END_STRUCT;
END_TYPE

TYPE "UDT_AHUsEqpDemandLimiter"
// stored: IsFailsafeCompliant false
   STRUCT
      rFan : Array[1..3] of Real;
      rExtractDumper : Array[1..3] of Real;
      rMixingDumper : Array[1..3] of Real;
      rHeater : Array[1..3] of Real;
      rCooler : Array[1..3] of Real;
      rWHU : Array[1..3] of Real;
   END_STRUCT;
END_TYPE

TYPE "UDT_AHUsMode"
// stored: IsFailsafeCompliant false
   STRUCT
      cPreviousOne { S7_SetPoint := 'True'} : Array[1..3] of Byte;
      cActual { S7_SetPoint := 'True'} : Array[1..3] of Byte;   // Поточний/Актуальний режим роботи
      cTarget { S7_SetPoint := 'True'} : Array[1..3] of Byte;   // Вибраний режим роботи, але ще не дійшли до нього
      cPreselectedOpModePLC : Array[1..3] of Byte;   // Вибор режиму роботи з PLC. 0-Protection/1-economy/2-PreComfort/3-Comfort/4-Auto
      cSchedulerTargetUnitOpMode : Array[1..3] of Byte;
      cPreselectedOpMode : Array[1..3] of Byte;   // Вибор режиму роботи з Фызичного перемикача на шафы. 0-Protection/1-economy/2-PreComfort/3-Comfort/4-Auto
   END_STRUCT;
END_TYPE

TYPE "UDT_AHUsFreshAirCoef"
// stored: IsFailsafeCompliant false
   STRUCT
      IAQ : Array[1..3] of Real;
      Temperature : Array[1..3] of Real;
      BuildingdP : Array[1..3] of Real;
   END_STRUCT;
   // Temperature[1..3] := 1.0;
END_TYPE

TYPE "UDT_AHUsRegulatorsDataType"
// stored: IsFailsafeCompliant false
   STRUCT
      cTempCooling : Array[1..3] of Byte;
      cTempHeating : Array[1..3] of Byte;
      cIAQ : Array[1..3] of Byte;
      cBuildingdP : Array[1..3] of Byte;
   END_STRUCT;
END_TYPE

TYPE "UDT_HSsDO"
// stored: IsFailsafeCompliant false
   STRUCT
      xBoilerEnable : Array[1..2] of Bool;
      xBoilerSt1Enable : Array[1..2] of Bool;
      xBoilerSt2Enable : Array[1..2] of Bool;
      xBoilerShuntPumpEnable : Array[1..2] of Bool;
      xBoilerShutOffValveCmd : Array[1..2] of Bool;
   END_STRUCT;
END_TYPE

TYPE "UDT_HCsAI"
// stored: IsFailsafeCompliant false
   STRUCT
      rSupplyWaterTemp : Array[1..2] of Real;
      rReturnWaterTemp : Array[1..2] of Real;
      r3vwPosFbk : Array[1..2] of Real;
   END_STRUCT;
END_TYPE

TYPE "UDT_HCsAO"
// stored: IsFailsafeCompliant false
   STRUCT
      rHC3vwCtrl : Array[1..2] of Real;
   END_STRUCT;
END_TYPE

TYPE "UDT_WSsAI"
// stored: IsFailsafeCompliant false
   STRUCT
      r14200a : Real;   // 14.200a
      r14201a : Real;   // 14.201a
   END_STRUCT;
END_TYPE

TYPE "UDT_ACsDO"
// stored: IsFailsafeCompliant false
   STRUCT
      xACCentralEnable : Bool;
   END_STRUCT;
END_TYPE

DATA_BLOCK "HVAC_Vars"   // DB99
{ S7_Optimized_Access := 'FALSE' }
VERSION : 0.1
// stored: AutoNumber false, DBAccessibleFromOPCUA true, IsOnlyStoredInLoadMemory false, IsWriteProtectedInAS false
   VAR
      Season { S7_SetPoint := 'True'} : "UDT_Store_Season";
      SetPoints { S7_SetPoint := 'True'} : "UDT_Store_Setpoints";
      OpModes { S7_SetPoint := 'True'} : "UDT_Store_OpMode";
      WeekScheduler { S7_SetPoint := 'True'} : "UDT_Store_Scheduler";
      RoomTempSetPointforHMI { S7_SetPoint := 'True'} : Real := 35.0;
      Holidays { S7_SetPoint := 'True'} : Array[1..4] of Date;
      xIsHoliday : Bool := FALSE;
      cDayType : Byte := 16#01;   // 0-WD,1-Mon,2-Cуб,3-Нед,4-Свят
      CurrentDate : Date := D#2026-04-20;
      CurrentTOD : Time_Of_Day := TOD#22:03:20.160;
      iRetVal : Int := 1;
   END_VAR
BEGIN
   Season.cSeasonModeSelection := 16#00;
   Season.cActual := 16#00;   // 0 = Summer 1 = Winter 2 = Midseason, 3=Auro
   Season.cTarget := 16#00;
   Season.cReserve := 16#00;
   Season.rOATtoWinter := 10.0;
   Season.rOATtoSummer := 12.0;
   SetPoints.Room.Actual.rRATHeating := 5.0;
   SetPoints.Room.Actual.rRATCooling := 35.0;
   SetPoints.Room.Actual.rIAQ := 0.0;
   SetPoints.Room.Actual.rBuildingdP := 0.0;
   SetPoints.Room.Comfort.rRATHeating := 18.0;
   SetPoints.Room.Comfort.rRATCooling := 22.0;
   SetPoints.Room.Comfort.rIAQ := 600.0;
   SetPoints.Room.Comfort.rBuildingdP := 5.0;
   SetPoints.Room.PreComfort.rRATHeating := 16.0;
   SetPoints.Room.PreComfort.rRATCooling := 25.0;
   SetPoints.Room.PreComfort.rIAQ := 800.0;
   SetPoints.Room.PreComfort.rBuildingdP := 2.0;
   SetPoints.Room.Econom.rRATHeating := 15.0;
   SetPoints.Room.Econom.rRATCooling := 30.0;
   SetPoints.Room.Econom.rIAQ := 0.0;
   SetPoints.Room.Econom.rBuildingdP := 0.0;
   SetPoints.Room.Protection.rRATHeating := 5.0;
   SetPoints.Room.Protection.rRATCooling := 35.0;
   SetPoints.Room.Protection.rIAQ := 0.0;
   SetPoints.Room.Protection.rBuildingdP := 0.0;
   OpModes.cPreviousOne := 16#00;
   OpModes.cActual := 16#00;
   OpModes.cTarget := 16#00;
   OpModes.cPreselectedOpMode := 16#00;
   WeekScheduler.cOpModeNowByScheduler := 16#02;   // 0 - Prot/ 1-Eco/ 2-PreComf/ 3- Comf/ 4 - Auto
   WeekScheduler.Monday.Comfort.Start := TOD#06:00:00;
   WeekScheduler.Monday.Comfort.Stop := TOD#21:00:00;
   WeekScheduler.Monday.PreComfort.Start := TOD#04:00:00;
   WeekScheduler.Monday.PreComfort.Stop := TOD#23:59:59;
   WeekScheduler.WorkingDays.Comfort.Start := TOD#06:00:00;
   WeekScheduler.WorkingDays.Comfort.Stop := TOD#21:00:00;
   WeekScheduler.WorkingDays.PreComfort.Start := TOD#00:00:00;
   WeekScheduler.WorkingDays.PreComfort.Stop := TOD#23:59:59;
   WeekScheduler.Saturday.Comfort.Start := TOD#06:00:00;
   WeekScheduler.Saturday.Comfort.Stop := TOD#21:00:00;
   WeekScheduler.Saturday.PreComfort.Start := TOD#00:00:00;
   WeekScheduler.Saturday.PreComfort.Stop := TOD#22:00:00;
   WeekScheduler.Sunday.Comfort.Start := TOD#06:00:00;
   WeekScheduler.Sunday.Comfort.Stop := TOD#18:00:00;
   WeekScheduler.Sunday.PreComfort.Start := TOD#05:30:00;
   WeekScheduler.Sunday.PreComfort.Stop := TOD#22:00:00;
   WeekScheduler.Holiday.Comfort.Start := TOD#00:00:00;
   WeekScheduler.Holiday.Comfort.Stop := TOD#00:00:00;
   WeekScheduler.Holiday.PreComfort.Start := TOD#00:00:00;
   WeekScheduler.Holiday.PreComfort.Stop := TOD#00:00:00;
   Holidays[1] := D#2026-01-01;
   Holidays[2] := D#2026-04-12;
   Holidays[3] := D#2027-01-01;
END_DATA_BLOCK

DATA_BLOCK "OAT"   // DB98
{ S7_Optimized_Access := 'FALSE' }
VERSION : 0.1
// stored: AutoNumber false, DBAccessibleFromOPCUA true, IsOnlyStoredInLoadMemory false, IsWriteProtectedInAS false
   VAR
      Temp { S7_SetPoint := 'True'} : "UDT_OAT";
      cSelectOATMode { S7_SetPoint := 'True'} : Byte;
   END_VAR
BEGIN
END_DATA_BLOCK

DATA_BLOCK "DL_Vars"   // DB51051
{ S7_Optimized_Access := 'FALSE'; DB_Accessible_From_OPC_UA := 'FALSE' }
VERSION : 0.1
// stored: AutoNumber false, DBAccessibleFromOPCUA false, IsOnlyStoredInLoadMemory false, IsWriteProtectedInAS false
   VAR
      Vars { S7_SetPoint := 'True'} : "UDT_DL_Vars";
   END_VAR
BEGIN
END_DATA_BLOCK

DATA_BLOCK "Timer"   // DB59999
{ S7_Optimized_Access := 'FALSE' }
VERSION : 0.1
// stored: AutoNumber false, DBAccessibleFromOPCUA true, IsOnlyStoredInLoadMemory false, IsWriteProtectedInAS false
   VAR
      x1SecRisingEdge : Bool;   // Одноразовий ымпуьс 1сек
      x1SecPrevClock : Bool;   // Попередный стан цикоу
      x1SecFired : Bool;   // Вже вiдпрацьовано?
   END_VAR
BEGIN
END_DATA_BLOCK

DATA_BLOCK "AHUDelays"   // DB110
{ S7_Optimized_Access := 'FALSE' }
VERSION : 0.1
// stored: AutoNumber false, DBAccessibleFromOPCUA true, IsOnlyStoredInLoadMemory false, IsWriteProtectedInAS false
   VAR RETAIN
      DelaysForStatus { S7_SetPoint := 'True'} : "UDT_AHUsStsDelay";
   END_VAR
BEGIN
END_DATA_BLOCK

DATA_BLOCK "AHUEqp"   // DB104
{ S7_Optimized_Access := 'FALSE' }
VERSION : 0.1
// stored: AutoNumber false, DBAccessibleFromOPCUA true, IsOnlyStoredInLoadMemory false, IsWriteProtectedInAS false
   VAR RETAIN
      Eqp { S7_SetPoint := 'True'} : "UDT_AHUEqp";
   END_VAR
BEGIN
   Eqp.Cfg.cFan[1] := 4;
   Eqp.Cfg.cFan[2] := 3;
   Eqp.Cfg.cExtractDumper[1] := 2;
   Eqp.Cfg.cMixingDumper[1..2] := 2;
   Eqp.Cfg.cHeater[1..2] := 2;
   Eqp.LimiterGridOperation.rFan[1..3] := 1.0;
   Eqp.LimiterGridOperation.rExtractDumper[1..3] := 1.0;
   Eqp.LimiterGridOperation.rMixingDumper[1..3] := 1.0;
   Eqp.LimiterGridOperation.rHeater[1..3] := 1.0;
   Eqp.LimiterGridOperation.rCooler[1..3] := 1.0;
   Eqp.LimiterGridOperation.rWHU[1..3] := 1.0;
   Eqp.LimiterDieselOperation.rFan[1..3] := 0.5;
   Eqp.LimiterDieselOperation.rExtractDumper[1..3] := 0.5;
   Eqp.LimiterDieselOperation.rMixingDumper[1..3] := 0.5;
   Eqp.LimiterDieselOperation.rHeater[1..3] := 1.0;
   Eqp.LimiterDieselOperation.rCooler[1..3] := 0.5;
   Eqp.LimiterDieselOperation.rWHU[1..3] := 1.0;
END_DATA_BLOCK

DATA_BLOCK "AHUFrostProt"   // DB109
{ S7_Optimized_Access := 'FALSE' }
VERSION : 0.1
// stored: AutoNumber false, DBAccessibleFromOPCUA true, IsOnlyStoredInLoadMemory false, IsWriteProtectedInAS false
   VAR RETAIN
      FrostProt { S7_SetPoint := 'True'} : "UDT_FrostProtection";
   END_VAR
BEGIN
   FrostProt.OATtoStartPreheating[1..3] := 10.0;
END_DATA_BLOCK

DATA_BLOCK "AHUOpModes"   // DB102
{ S7_Optimized_Access := 'FALSE' }
VERSION : 0.1
// stored: AutoNumber false, DBAccessibleFromOPCUA true, IsOnlyStoredInLoadMemory false, IsWriteProtectedInAS false
   VAR RETAIN
      OpModes { S7_SetPoint := 'True'} : "UDT_AHUsMode";
   END_VAR
BEGIN
   OpModes.cPreselectedOpModePLC[1..3] := 0;
   OpModes.cSchedulerTargetUnitOpMode[1..2] := 3;
   OpModes.cSchedulerTargetUnitOpMode[3] := 0;
END_DATA_BLOCK

DATA_BLOCK "AHURegulators"   // DB105
{ S7_Optimized_Access := 'FALSE' }
VERSION : 0.1
// stored: AutoNumber false, DBAccessibleFromOPCUA true, IsOnlyStoredInLoadMemory false, IsWriteProtectedInAS false
   VAR RETAIN
      Regulators { S7_SetPoint := 'True'} : "UDT_AHUsRegulators";
   END_VAR
BEGIN
   Regulators.Cfg.cTempHeating[1] := 2;
   Regulators.FreshAirCoef.IAQ[1..3] := 0.2;
   Regulators.FreshAirCoef.BuildingdP[1..3] := 0.2;
END_DATA_BLOCK

DATA_BLOCK "AHUSetPoints"   // DB106
{ S7_Optimized_Access := 'FALSE' }
VERSION : 0.1
// stored: AutoNumber false, DBAccessibleFromOPCUA true, IsOnlyStoredInLoadMemory false, IsWriteProtectedInAS false
   VAR RETAIN
      SetPoints { S7_SetPoint := 'True'} : "UDT_AHUSetpoints";
   END_VAR
BEGIN
END_DATA_BLOCK

DATA_BLOCK "AHUSustained"   // DB115
{ S7_Optimized_Access := 'FALSE' }
VERSION : 0.1
// stored: AutoNumber false, DBAccessibleFromOPCUA true, IsOnlyStoredInLoadMemory false, IsWriteProtectedInAS false
   VAR RETAIN
      Requests { S7_SetPoint := 'True'} : "UDT_AHUsSustainedRequests";
   END_VAR
BEGIN
END_DATA_BLOCK

DATA_BLOCK "AHUUnitStates"   // DB103
{ S7_Optimized_Access := 'FALSE' }
VERSION : 0.1
// stored: AutoNumber false, DBAccessibleFromOPCUA true, IsOnlyStoredInLoadMemory false, IsWriteProtectedInAS false
   VAR RETAIN
      UnitStates { S7_SetPoint := 'True'} : "UDT_AHUsState";
   END_VAR
BEGIN
   UnitStates.cPreviousOne[1..2] := 0;
END_DATA_BLOCK

DATA_BLOCK "BoilerOnOffSettings"   // DB1017
{ S7_Optimized_Access := 'FALSE' }
VERSION : 0.1
// stored: AutoNumber false, DBAccessibleFromOPCUA true, IsOnlyStoredInLoadMemory false, IsWriteProtectedInAS false
   VAR
      Boiler { S7_SetPoint := 'True'} : "UDT_BoilersOnOffSettings";
   END_VAR
BEGIN
   Boiler.PLCModeSelection.cPreselectedOpModePLC := 16#3;
   Boiler.PLCModeSelection.cActualOpModePLC := 16#3;
END_DATA_BLOCK

DATA_BLOCK "HSSetPoints"   // DB1019
{ S7_Optimized_Access := 'FALSE' }
VERSION : 0.1
// stored: AutoNumber false, DBAccessibleFromOPCUA true, IsOnlyStoredInLoadMemory false, IsWriteProtectedInAS false
   VAR RETAIN
      SetPoints { S7_SetPoint := 'True'} : "UDT_AHUSetpoints";
   END_VAR
BEGIN
END_DATA_BLOCK

DATA_BLOCK "DHWAI"   // DB1400
{ S7_Optimized_Access := 'FALSE' }
VERSION : 0.1
// stored: AutoNumber false, DBAccessibleFromOPCUA true, IsOnlyStoredInLoadMemory false, IsWriteProtectedInAS false
   VAR
      AI { S7_SetPoint := 'True'} : "UDT_WSsAI";
   END_VAR
BEGIN
END_DATA_BLOCK

DATA_BLOCK "HCsAO"   // DB1023
{ S7_Optimized_Access := 'FALSE' }
VERSION : 0.1
// stored: AutoNumber false, DBAccessibleFromOPCUA true, IsOnlyStoredInLoadMemory false, IsWriteProtectedInAS false
   VAR
      AO { S7_SetPoint := 'True'} : "UDT_HCsAO";
   END_VAR
BEGIN
END_DATA_BLOCK

DATA_BLOCK "HCsDI"   // DB1024
{ S7_Optimized_Access := 'FALSE' }
VERSION : 0.1
// stored: AutoNumber false, DBAccessibleFromOPCUA true, IsOnlyStoredInLoadMemory false, IsWriteProtectedInAS false
   VAR
      Requests { S7_SetPoint := 'True'} : "UDT_HCsDI";
   END_VAR
BEGIN
END_DATA_BLOCK

DATA_BLOCK "HCsDO"   // DB1022
{ S7_Optimized_Access := 'FALSE' }
VERSION : 0.1
// stored: AutoNumber false, DBAccessibleFromOPCUA true, IsOnlyStoredInLoadMemory false, IsWriteProtectedInAS false
   VAR
      Requests { S7_SetPoint := 'True'} : "UDT_HCsDO";
   END_VAR
BEGIN
END_DATA_BLOCK

DATA_BLOCK "HSsAI"   // DB1021
{ S7_Optimized_Access := 'FALSE' }
VERSION : 0.1
// stored: AutoNumber false, DBAccessibleFromOPCUA true, IsOnlyStoredInLoadMemory false, IsWriteProtectedInAS false
   VAR
      AI : "UDT_HSsAI";
   END_VAR
BEGIN
END_DATA_BLOCK

DATA_BLOCK "HSsDI"   // DB1025
{ S7_Optimized_Access := 'FALSE' }
VERSION : 0.1
// stored: AutoNumber false, DBAccessibleFromOPCUA true, IsOnlyStoredInLoadMemory false, IsWriteProtectedInAS false
   VAR
      Requests { S7_SetPoint := 'True'} : "UDT_HSsDI";
   END_VAR
BEGIN
END_DATA_BLOCK

DATA_BLOCK "HSsDO"   // DB1028
{ S7_Optimized_Access := 'FALSE' }
VERSION : 0.1
// stored: AutoNumber false, DBAccessibleFromOPCUA true, IsOnlyStoredInLoadMemory false, IsWriteProtectedInAS false
   VAR
      Requests { S7_SetPoint := 'True'} : "UDT_HSsDO";
   END_VAR
BEGIN
END_DATA_BLOCK

DATA_BLOCK "AHUAO"   // DB112
{ S7_Optimized_Access := 'FALSE' }
VERSION : 0.1
// stored: AutoNumber false, DBAccessibleFromOPCUA true, IsOnlyStoredInLoadMemory false, IsWriteProtectedInAS false
   VAR
      AO { S7_SetPoint := 'True'} : "UTD_AHUsAO";
   END_VAR
BEGIN
END_DATA_BLOCK

DATA_BLOCK "AHUDI"   // DB113
{ S7_Optimized_Access := 'FALSE' }
VERSION : 0.1
// stored: AutoNumber false, DBAccessibleFromOPCUA true, IsOnlyStoredInLoadMemory false, IsWriteProtectedInAS false
   VAR RETAIN
      DI { S7_SetPoint := 'True'} : "UDT_AHUsDI";
   END_VAR
BEGIN
END_DATA_BLOCK

DATA_BLOCK "AHUDO"   // DB114
{ S7_Optimized_Access := 'FALSE' }
VERSION : 0.1
// stored: AutoNumber false, DBAccessibleFromOPCUA true, IsOnlyStoredInLoadMemory false, IsWriteProtectedInAS false
   VAR
      Requests { S7_SetPoint := 'True'} : "UDT_AHUsDO";
   END_VAR
BEGIN
END_DATA_BLOCK

DATA_BLOCK "DLsDI"   // DB51025
{ S7_Optimized_Access := 'FALSE' }
VERSION : 0.1
// stored: AutoNumber false, DBAccessibleFromOPCUA true, IsOnlyStoredInLoadMemory false, IsWriteProtectedInAS false
   VAR
      Requests : "UDT_DLsDI";
   END_VAR
BEGIN
END_DATA_BLOCK

DATA_BLOCK "ACDO"   // DB724
{ S7_Optimized_Access := 'FALSE' }
VERSION : 0.1
// stored: AutoNumber false, DBAccessibleFromOPCUA true, IsOnlyStoredInLoadMemory false, IsWriteProtectedInAS false
   VAR
      Requests : "UDT_ACsDO";
   END_VAR
BEGIN
END_DATA_BLOCK

DATA_BLOCK "AHDO"   // DB824
{ S7_Optimized_Access := 'FALSE' }
VERSION : 0.1
// stored: AutoNumber false, DBAccessibleFromOPCUA true, IsOnlyStoredInLoadMemory false, IsWriteProtectedInAS false
   VAR
      Requests : "UDT_AHsDO";
   END_VAR
BEGIN
END_DATA_BLOCK

DATA_BLOCK "DLsAI"   // DB51021
{ S7_Optimized_Access := 'FALSE' }
VERSION : 0.1
// stored: AutoNumber false, DBAccessibleFromOPCUA true, IsOnlyStoredInLoadMemory false, IsWriteProtectedInAS false
   VAR
      AI : "UDT_DLsAI";
   END_VAR
BEGIN
   AI.rDayTankLevel[1] := 0.0;
END_DATA_BLOCK

DATA_BLOCK "DLsDO"   // DB51028
{ S7_Optimized_Access := 'FALSE' }
VERSION : 0.1
// stored: AutoNumber false, DBAccessibleFromOPCUA true, IsOnlyStoredInLoadMemory false, IsWriteProtectedInAS false
   VAR
      Requests : "UDT_DLsDO";
   END_VAR
BEGIN
END_DATA_BLOCK

DATA_BLOCK "AHUProxyCH"   // DB59021
{ S7_Optimized_Access := 'FALSE' }
VERSION : 0.1
// stored: AutoNumber false, DBAccessibleFromOPCUA true, IsOnlyStoredInLoadMemory false, IsWriteProtectedInAS false
   VAR
      Vars { S7_SetPoint := 'True'} : "UDT_AnalogProxyCH_Vars";
   END_VAR
BEGIN
END_DATA_BLOCK

DATA_BLOCK "AHUAlarms"   // DB101
{ S7_Optimized_Access := 'FALSE' }
VERSION : 0.1
// stored: AutoNumber false, DBAccessibleFromOPCUA true, IsOnlyStoredInLoadMemory false, IsWriteProtectedInAS false
   VAR
      Summary { S7_SetPoint := 'True'} : "UDT_AHUSummaryAlarms";
   END_VAR
BEGIN
END_DATA_BLOCK

DATA_BLOCK "AHUAI"   // DB111
{ S7_Optimized_Access := 'FALSE' }
VERSION : 0.1
// stored: AutoNumber false, DBAccessibleFromOPCUA true, IsOnlyStoredInLoadMemory false, IsWriteProtectedInAS false
   VAR
      AI { S7_SetPoint := 'True'} : "UDT_AHUsAI";
   END_VAR
BEGIN
   AI.rIAQ[1..3] := 0.0;
   AI.rBuildingdP[1..3] := 0.0;
   AI.rRoomAirTemp_PLC_AI[1..3] := 0.0;
   AI.rSupplyAirTemp[1] := 26.69;
   AI.rSupplyAirTemp[2] := 0.0;
   AI.rSupplyAirTemp[3] := 22.39;
   AI.rReturnAirTemp[1..3] := 0.0;
   AI.rFrostProtWaterTemp[1] := 3276.7;
   AI.rFrostProtWaterTemp[2] := 0.0;
   AI.rFrostProtWaterTemp[3] := 21.31;
   AI.rFrostProtAirTemp[1] := 17.07954;
   AI.rFrostProtAirTemp[2..3] := 0.0;
   AI.rRoomAirRelHumi[1..2] := 0.0;
   AI.rRoomAirRelHumi[3] := 21.23;
   AI.rReserve[1..3] := 0.0;
   AI.rSAFilterdP[1] := 5.714699;
   AI.rSAFilterdP[2..3] := 0.0;
   AI.cRoomTempSelect[1] := 2;
END_DATA_BLOCK

DATA_BLOCK "BoilerAlarms"   // DB1015
{ S7_Optimized_Access := 'TRUE' }
VERSION : 0.1
// stored: AutoNumber false, DBAccessibleFromOPCUA true, IsOnlyStoredInLoadMemory false, IsRetainMemResEnabled false, IsWriteProtectedInAS false, MemoryReserve 100
   VAR
      Summary { S7_SetPoint := 'True'} : "UDT_BoilersSummaryAlarms";
   END_VAR
BEGIN
END_DATA_BLOCK

DATA_BLOCK "BoilerOpModes"   // DB1016
{ S7_Optimized_Access := 'FALSE' }
VERSION : 0.1
// stored: AutoNumber false, DBAccessibleFromOPCUA true, IsOnlyStoredInLoadMemory false, IsWriteProtectedInAS false
   VAR
      OpModes { S7_SetPoint := 'True'} : "UDT_BoilerOpMode";
   END_VAR
BEGIN
END_DATA_BLOCK

DATA_BLOCK "BoilerUnitStates"   // DB1
{ S7_Optimized_Access := 'TRUE' }
VERSION : 0.1
// stored: AutoNumber true, DBAccessibleFromOPCUA true, IsOnlyStoredInLoadMemory false, IsRetainMemResEnabled false, IsWriteProtectedInAS false, MemoryReserve 100
   VAR
      UnitStates { S7_SetPoint := 'True'} : "UDT_BoilerUnitState";
   END_VAR
BEGIN
END_DATA_BLOCK

DATA_BLOCK "Vitogate"   // DB1010
{ S7_Optimized_Access := 'FALSE' }
VERSION : 0.1
// stored: AutoNumber false, DBAccessibleFromOPCUA true, IsOnlyStoredInLoadMemory false, IsWriteProtectedInAS false
   VAR
      Alarms { S7_SetPoint := 'True'} : "UDT_Vitotronic100_Alarms";
      IOs { S7_SetPoint := 'True'} : "UDT_Vitotronic100_IOs";
      Params { S7_SetPoint := 'True'} : "UDT_Vitotronic100_Params";
      Settings { S7_SetPoint := 'True'} : "UDT_Vitotronic100_Settings";
   END_VAR
BEGIN
END_DATA_BLOCK

DATA_BLOCK "WeatherComp"   // DB1018
{ S7_Optimized_Access := 'FALSE' }
VERSION : 0.1
// stored: AutoNumber false, DBAccessibleFromOPCUA true, IsOnlyStoredInLoadMemory false, IsWriteProtectedInAS false
   VAR
      WeatherComp { S7_SetPoint := 'True'} : "UDT_WeatherCompCurve";
   END_VAR
BEGIN
END_DATA_BLOCK

DATA_BLOCK "HCsAI"   // DB1020
{ S7_Optimized_Access := 'FALSE' }
VERSION : 0.1
// stored: AutoNumber false, DBAccessibleFromOPCUA true, IsOnlyStoredInLoadMemory false, IsWriteProtectedInAS false
   VAR
      AI { S7_SetPoint := 'True'} : "UDT_HCsAI";
   END_VAR
BEGIN
END_DATA_BLOCK

DATA_BLOCK "Boilers"   // DB1030
{ S7_Optimized_Access := 'FALSE' }
VERSION : 0.1
// stored: AutoNumber false, DBAccessibleFromOPCUA true, IsOnlyStoredInLoadMemory false, IsWriteProtectedInAS false
   VAR
      Boilers { S7_SetPoint := 'True'} : "UDT_BoilerUnitState";
   END_VAR
BEGIN
END_DATA_BLOCK

DATA_BLOCK "SS1_CPU1215_AI_Vars"   // DB11011
{ S7_Optimized_Access := 'FALSE' }
VERSION : 0.1
// stored: AutoNumber false, DBAccessibleFromOPCUA true, IsOnlyStoredInLoadMemory false, IsWriteProtectedInAS false
   VAR
      AI1 { S7_SetPoint := 'True'} : "UDT_AIadv";
      AI2 { S7_SetPoint := 'True'} : "UDT_AIadv";
   END_VAR
BEGIN
   AI1.rValue := 368.9236;
   AI1.rMin := 0.0;
   AI1.rMax := 50000.0;
   AI1.rCalibration := 0.0;
   AI1.iFuncSystemID := 16#01;
   AI1.iFuncVar := 16#0B;
   AI1.rFilterSet := 0.0;
   AI2.rValue := 0.0;
   AI2.rMin := 0.0;
   AI2.rMax := 0.0;
   AI2.rCalibration := 0.0;
   AI2.iFuncSystemID := 16#00;
   AI2.iFuncVar := 16#00;
   AI2.rFilterSet := 0.0;
END_DATA_BLOCK

DATA_BLOCK "SS1_CPU1215_AO_Vars"   // DB11012
{ S7_Optimized_Access := 'FALSE' }
VERSION : 0.1
// stored: AutoNumber false, DBAccessibleFromOPCUA true, IsOnlyStoredInLoadMemory false, IsWriteProtectedInAS false
   VAR
      AO1 { S7_SetPoint := 'True'} : "UDT_AOadv";
      AO2 { S7_SetPoint := 'True'} : "UDT_AOadv";
   END_VAR
BEGIN
   AO1.rInput := 0.0;
   AO1.cMOA := 16#01;
   AO1.cFuncSystemID := 1;
   AO1.cFuncVar := 1;
   AO1.cMemory := 16#00;
   AO1.rManOutput := 60.0;
   AO1.iOutput := 11060;
   AO2.rInput := 0.0;
   AO2.cMOA := 16#00;
   AO2.cFuncSystemID := 16#00;
   AO2.cFuncVar := 16#00;
   AO2.cMemory := 16#00;
   AO2.rManOutput := 0.0;
   AO2.iOutput := 0;
END_DATA_BLOCK

DATA_BLOCK "SS1_CPU1215_DI_Vars"   // DB11013
{ S7_Optimized_Access := 'FALSE' }
VERSION : 0.1
// stored: AutoNumber false, DBAccessibleFromOPCUA true, IsOnlyStoredInLoadMemory false, IsWriteProtectedInAS false
   VAR
      DI1 : "UDT_DIadv";
      DI2 : "UDT_DIadv";
      DI3 : "UDT_DIadv";
      DI4 : "UDT_DIadv";
      DI5 : "UDT_DIadv";
      DI6 : "UDT_DIadv";
      DI7 { S7_SetPoint := 'True'} : "UDT_DIadv";
      DI8 { S7_SetPoint := 'True'} : "UDT_DIadv";
      DI9 { S7_SetPoint := 'True'} : "UDT_DIadv";
      DI10 { S7_SetPoint := 'True'} : "UDT_DIadv";
      DI11 { S7_SetPoint := 'True'} : "UDT_DIadv";
      DI12 { S7_SetPoint := 'True'} : "UDT_DIadv";
      DI13 { S7_SetPoint := 'True'} : "UDT_DIadv";
      DI14 { S7_SetPoint := 'True'} : "UDT_DIadv";
   END_VAR
BEGIN
   DI1.cFuncSystemID := 3;
   DI1.cFuncVar := 19;
   DI2.cFuncSystemID := 3;
   DI2.cFuncVar := 8;
   DI3.cFuncSystemID := 3;
   DI3.cFuncVar := 9;
   DI4.cFuncSystemID := 3;
   DI4.cFuncVar := 20;
   DI5.cFuncSystemID := 3;
   DI5.cFuncVar := 7;
   DI6.cFuncSystemID := 3;
   DI6.cFuncVar := 21;
   DI8.cFuncSystemID := 10;
   DI8.cFuncVar := 41;
   DI9.cFuncSystemID := 10;
   DI9.cFuncVar := 43;
   DI10.cFuncSystemID := 3;
   DI10.cFuncVar := 16;
   DI11.cFuncSystemID := 3;
   DI11.cFuncVar := 18;
   DI12.cFuncSystemID := 10;
   DI12.cFuncVar := 29;
   DI13.cFuncSystemID := 10;
   DI13.cFuncVar := 28;
END_DATA_BLOCK

DATA_BLOCK "SS1_CPU1215_DO_Vars"   // DB11014
{ S7_Optimized_Access := 'FALSE' }
VERSION : 0.1
// stored: AutoNumber false, DBAccessibleFromOPCUA true, IsOnlyStoredInLoadMemory false, IsWriteProtectedInAS false
   VAR
      DO1 { S7_SetPoint := 'True'} : "UDT_DOadv";
      DO2 { S7_SetPoint := 'True'} : "UDT_DOadv";
      DO3 { S7_SetPoint := 'True'} : "UDT_DOadv";
      DO4 { S7_SetPoint := 'True'} : "UDT_DOadv";
      DO5 { S7_SetPoint := 'True'} : "UDT_DOadv";
      DO6 : "UDT_DOadv";
      DO7 { S7_SetPoint := 'True'} : "UDT_DOadv";
      DO8 { S7_SetPoint := 'True'} : "UDT_DOadv";
      DO9 { S7_SetPoint := 'True'} : "UDT_DOadv";
      DO10 { S7_SetPoint := 'True'} : "UDT_DOadv";
   END_VAR
BEGIN
END_DATA_BLOCK

DATA_BLOCK "SS1_A2_8RTD_AI_Vars"   // DB11021
{ S7_Optimized_Access := 'FALSE' }
VERSION : 0.1
// stored: AutoNumber false, DBAccessibleFromOPCUA true, IsOnlyStoredInLoadMemory false, IsWriteProtectedInAS false
   VAR
      AI1 { S7_SetPoint := 'True'} : "UDT_RTDadv";
      AI2 { S7_SetPoint := 'True'} : "UDT_RTDadv";
      AI3 { S7_SetPoint := 'True'} : "UDT_RTDadv";
      AI4 { S7_SetPoint := 'True'} : "UDT_RTDadv";
      AI5 { S7_SetPoint := 'True'} : "UDT_RTDadv";
      AI6 { S7_SetPoint := 'True'} : "UDT_RTDadv";
      AI7 { S7_SetPoint := 'True'} : "UDT_RTDadv";
      AI8 { S7_SetPoint := 'True'} : "UDT_RTDadv";
   END_VAR
BEGIN
   AI1.rValue := 26.03;
   AI1.rFilterSet := 0.0;
   AI1.rCalibration := 0.0;
   AI1.rDiv := 100.0;
   AI1.cFuncSystemID := 10;
   AI1.cFuncVar := 4;
   AI1.iReserv := 0;
   AI2.rValue := 3276.7;
   AI2.rFilterSet := 0.0;
   AI2.rCalibration := 0.0;
   AI2.rDiv := 10.0;
   AI2.cFuncSystemID := 16#01;
   AI2.cFuncVar := 16#06;
   AI2.iReserv := 0;
   AI3.rValue := 26.7;
   AI3.rFilterSet := 0.0;
   AI3.rCalibration := 0.0;
   AI3.rDiv := 100.0;
   AI3.cFuncSystemID := 16#01;
   AI3.cFuncVar := 16#04;
   AI3.iReserv := 0;
   AI4.rValue := 22.39;
   AI4.rFilterSet := 0.0;
   AI4.rCalibration := 0.0;
   AI4.rDiv := 100.0;
   AI4.cFuncSystemID := 16#03;
   AI4.cFuncVar := 16#04;
   AI4.iReserv := 0;
   AI5.rValue := 24.7;
   AI5.rFilterSet := 0.0;
   AI5.rCalibration := 0.0;
   AI5.rDiv := 10.0;
   AI5.cFuncSystemID := 16#0A;
   AI5.cFuncVar := 16#01;
   AI5.iReserv := 0;
   AI6.rValue := 61.78;
   AI6.rFilterSet := 0.0;
   AI6.rCalibration := 0.0;
   AI6.rDiv := 100.0;
   AI6.cFuncSystemID := 16#0E;
   AI6.cFuncVar := 16#01;
   AI6.iReserv := 0;
   AI7.rValue := 28.62;
   AI7.rFilterSet := 0.0;
   AI7.rCalibration := 0.0;
   AI7.rDiv := 100.0;
   AI7.cFuncSystemID := 16#0E;
   AI7.cFuncVar := 16#02;
   AI7.iReserv := 0;
   AI8.rValue := 21.31;
   AI8.rFilterSet := 0.0;
   AI8.rCalibration := 0.0;
   AI8.rDiv := 100.0;
   AI8.cFuncSystemID := 16#03;
   AI8.cFuncVar := 16#06;
   AI8.iReserv := 0;
END_DATA_BLOCK

DATA_BLOCK "SS1_A3_8xAI_AI_Vars"   // DB11031
{ S7_Optimized_Access := 'FALSE' }
VERSION : 0.1
// stored: AutoNumber false, DBAccessibleFromOPCUA true, IsOnlyStoredInLoadMemory false, IsWriteProtectedInAS false
   VAR
      AI1 { S7_SetPoint := 'True'} : "UDT_AIadv";
      AI2 { S7_SetPoint := 'True'} : "UDT_AIadv";
      AI3 { S7_SetPoint := 'True'} : "UDT_AIadv";
      AI4 { S7_SetPoint := 'True'} : "UDT_AIadv";
      AI5 { S7_SetPoint := 'True'} : "UDT_AIadv";
      AI6 { S7_SetPoint := 'True'} : "UDT_AIadv";
      AI7 { S7_SetPoint := 'True'} : "UDT_AIadv";
      AI8 { S7_SetPoint := 'True'} : "UDT_AIadv";
   END_VAR
BEGIN
   AI1.rValue := 0.3255208;
   AI1.rMin := 0.0;
   AI1.rMax := 1000.0;
   AI1.rCalibration := 0.0;
   AI1.iFuncSystemID := 16#00;
   AI1.iFuncVar := 16#00;
   AI1.rFilterSet := 0.0;
   AI2.rValue := 1.808449;
   AI2.rMin := 0.0;
   AI2.rMax := 1000.0;
   AI2.rCalibration := 0.0;
   AI2.iFuncSystemID := 16#00;
   AI2.iFuncVar := 16#00;
   AI2.rFilterSet := 0.0;
   AI3.rValue := 3.616898E-05;
   AI3.rMin := 0.0;
   AI3.rMax := 0.0;
   AI3.rCalibration := 0.0;
   AI3.iFuncSystemID := 16#00;
   AI3.iFuncVar := 16#00;
   AI3.rFilterSet := 0.0;
   AI4.rValue := 0.0003255208;
   AI4.rMin := 0.0;
   AI4.rMax := 0.0;
   AI4.rCalibration := 0.0;
   AI4.iFuncSystemID := 16#00;
   AI4.iFuncVar := 16#00;
   AI4.rFilterSet := 0.0;
   AI5.rValue := 6.04022;
   AI5.rMin := 0.0;
   AI5.rMax := 1000.0;
   AI5.rCalibration := 0.0;
   AI5.iFuncSystemID := 16#01;
   AI5.iFuncVar := 16#0A;
   AI5.rFilterSet := 0.0;
   AI6.rValue := 17.15549;
   AI6.rMin := 0.0;
   AI6.rMax := 15.0;
   AI6.rCalibration := 0.0;
   AI6.iFuncSystemID := 16#01;
   AI6.iFuncVar := 16#07;
   AI6.rFilterSet := 0.0;
   AI7.rValue := 29.49942;
   AI7.rMin := 0.0;
   AI7.rMax := 100.0;
   AI7.rCalibration := 0.0;
   AI7.iFuncSystemID := 16#00;
   AI7.iFuncVar := 16#00;
   AI7.rFilterSet := 0.0;
   AI8.rValue := 0.07957176;
   AI8.rMin := 0.0;
   AI8.rMax := 100.0;
   AI8.rCalibration := 0.0;
   AI8.iFuncSystemID := 16#00;
   AI8.iFuncVar := 16#00;
   AI8.rFilterSet := 0.0;
END_DATA_BLOCK

DATA_BLOCK "SS1_A4_4AO_AO_Vars"   // DB11041
{ S7_Optimized_Access := 'FALSE' }
VERSION : 0.1
// stored: AutoNumber false, DBAccessibleFromOPCUA true, IsOnlyStoredInLoadMemory false, IsWriteProtectedInAS false
   VAR
      AO1 { S7_SetPoint := 'True'} : "UDT_AOadv";
      AO2 { S7_SetPoint := 'True'} : "UDT_AOadv";
      AO3 : "UDT_AOadv";
      AO4 : "UDT_AOadv";
   END_VAR
BEGIN
   AO1.cFuncSystemID := 1;
   AO1.cFuncVar := 2;
   AO2.cFuncSystemID := 1;
   AO2.cFuncVar := 3;
   AO3.cFuncSystemID := 3;
   AO3.cFuncVar := 2;
   AO4.cFuncSystemID := 1;
   AO4.cFuncVar := 4;
END_DATA_BLOCK

DATA_BLOCK "SS1_A5_16DI_DI_Vars"   // DB11051
{ S7_Optimized_Access := 'FALSE' }
VERSION : 0.1
// stored: AutoNumber false, DBAccessibleFromOPCUA true, IsOnlyStoredInLoadMemory false, IsWriteProtectedInAS false
   VAR
      DI1 : "UDT_DIadv";
      DI2 : "UDT_DIadv";
      DI3 : "UDT_DIadv";
      DI4 : "UDT_DIadv";
      DI5 : "UDT_DIadv";
      DI6 : "UDT_DIadv";
      DI7 : "UDT_DIadv";
      DI8 : "UDT_DIadv";
      DI9 { S7_SetPoint := 'True'} : "UDT_DIadv";
      DI10 { S7_SetPoint := 'True'} : "UDT_DIadv";
      DI11 { S7_SetPoint := 'True'} : "UDT_DIadv";
      DI12 { S7_SetPoint := 'True'} : "UDT_DIadv";
      DI13 { S7_SetPoint := 'True'} : "UDT_DIadv";
      DI14 { S7_SetPoint := 'True'} : "UDT_DIadv";
      DI15 { S7_SetPoint := 'True'} : "UDT_DIadv";
      DI16 { S7_SetPoint := 'True'} : "UDT_DIadv";
   END_VAR
BEGIN
   DI3.cFuncSystemID := 10;
   DI3.cFuncVar := 25;
   DI4.cFuncSystemID := 10;
   DI4.cFuncVar := 26;
   DI5.cFuncSystemID := 10;
   DI5.cFuncVar := 27;
   DI6.cFuncSystemID := 100;
   DI6.cFuncVar := 11;
   DI7.cFuncSystemID := 100;
   DI7.cFuncVar := 12;
   DI8.cFuncSystemID := 10;
   DI8.cFuncVar := 24;
   DI9.cFuncSystemID := 10;
   DI9.cFuncVar := 22;
   DI10.xInversion := true;
   DI10.cFuncSystemID := 10;
   DI10.cFuncVar := 23;
   DI11.cFuncSystemID := 10;
   DI11.cFuncVar := 7;
   DI12.cFuncSystemID := 10;
   DI12.cFuncVar := 2;
   DI13.xInversion := true;
   DI13.cFuncSystemID := 10;
   DI13.cFuncVar := 3;
   DI14.cFuncSystemID := 10;
   DI14.cFuncVar := 5;
   DI15.xInversion := true;
   DI15.cFuncSystemID := 10;
   DI15.cFuncVar := 6;
END_DATA_BLOCK

DATA_BLOCK "SS1_A6_16DI_DI_Vars"   // DB11061
{ S7_Optimized_Access := 'FALSE' }
VERSION : 0.1
// stored: AutoNumber false, DBAccessibleFromOPCUA true, IsOnlyStoredInLoadMemory false, IsWriteProtectedInAS false
   VAR
      DI1 : "UDT_DIadv";
      DI2 : "UDT_DIadv";
      DI3 : "UDT_DIadv";
      DI4 : "UDT_DIadv";
      DI5 : "UDT_DIadv";
      DI6 : "UDT_DIadv";
      DI7 : "UDT_DIadv";
      DI8 : "UDT_DIadv";
      DI9 { S7_SetPoint := 'True'} : "UDT_DIadv";
      DI10 { S7_SetPoint := 'True'} : "UDT_DIadv";
      DI11 { S7_SetPoint := 'True'} : "UDT_DIadv";
      DI12 { S7_SetPoint := 'True'} : "UDT_DIadv";
      DI13 { S7_SetPoint := 'True'} : "UDT_DIadv";
      DI14 { S7_SetPoint := 'True'} : "UDT_DIadv";
      DI15 { S7_SetPoint := 'True'} : "UDT_DIadv";
      DI16 { S7_SetPoint := 'True'} : "UDT_DIadv";
   END_VAR
BEGIN
   DI1.cFuncSystemID := 100;
   DI1.cFuncVar := 1;
   DI2.cFuncSystemID := 100;
   DI2.cFuncVar := 3;
   DI5.cFuncSystemID := 100;
   DI5.cFuncVar := 5;
   DI6.cFuncSystemID := 100;
   DI6.cFuncVar := 6;
END_DATA_BLOCK

DATA_BLOCK "SS1_A7_16DI_16DO_DI_Vars"   // DB11071
{ S7_Optimized_Access := 'FALSE' }
VERSION : 0.1
// stored: AutoNumber false, DBAccessibleFromOPCUA true, IsOnlyStoredInLoadMemory false, IsWriteProtectedInAS false
   VAR
      DI1 : "UDT_DIadv";
      DI2 : "UDT_DIadv";
      DI3 : "UDT_DIadv";
      DI4 : "UDT_DIadv";
      DI5 : "UDT_DIadv";
      DI6 : "UDT_DIadv";
      DI7 : "UDT_DIadv";
      DI8 : "UDT_DIadv";
      DI9 { S7_SetPoint := 'True'} : "UDT_DIadv";
      DI10 { S7_SetPoint := 'True'} : "UDT_DIadv";
      DI11 { S7_SetPoint := 'True'} : "UDT_DIadv";
      DI12 { S7_SetPoint := 'True'} : "UDT_DIadv";
      DI13 { S7_SetPoint := 'True'} : "UDT_DIadv";
      DI14 { S7_SetPoint := 'True'} : "UDT_DIadv";
      DI15 { S7_SetPoint := 'True'} : "UDT_DIadv";
      DI16 { S7_SetPoint := 'True'} : "UDT_DIadv";
   END_VAR
BEGIN
   DI4.cFuncSystemID := 100;
   DI4.cFuncVar := 7;
   DI5.cFuncSystemID := 1;
   DI5.cFuncVar := 17;
   DI6.cFuncSystemID := 1;
   DI6.cFuncVar := 18;
   DI7.cFuncSystemID := 1;
   DI7.cFuncVar := 16;
   DI9.cFuncSystemID := 1;
   DI10.cFuncSystemID := 1;
   DI10.cFuncVar := 2;
   DI11.cFuncSystemID := 1;
   DI11.cFuncVar := 3;
   DI12.cFuncSystemID := 1;
   DI13.cFuncSystemID := 1;
   DI13.cFuncVar := 14;
   DI14.cFuncSystemID := 1;
   DI15.cFuncSystemID := 1;
   DI15.cFuncVar := 19;
   DI16.cFuncSystemID := 1;
   DI16.cFuncVar := 8;
END_DATA_BLOCK

DATA_BLOCK "SS1_A7_16DI_16DO_DO_Vars"   // DB11072
{ S7_Optimized_Access := 'FALSE' }
VERSION : 0.1
// stored: AutoNumber false, DBAccessibleFromOPCUA true, IsOnlyStoredInLoadMemory false, IsWriteProtectedInAS false
   VAR
      DO1 { S7_SetPoint := 'True'} : "UDT_DOadv";
      DO2 { S7_SetPoint := 'True'} : "UDT_DOadv";
      DO3 { S7_SetPoint := 'True'} : "UDT_DOadv";
      DO4 { S7_SetPoint := 'True'} : "UDT_DOadv";
      DO5 { S7_SetPoint := 'True'} : "UDT_DOadv";
      DO6 { S7_SetPoint := 'True'} : "UDT_DOadv";
      DO7 { S7_SetPoint := 'True'} : "UDT_DOadv";
      DO8 { S7_SetPoint := 'True'} : "UDT_DOadv";
      DO9 { S7_SetPoint := 'True'} : "UDT_DOadv";
      DO10 { S7_SetPoint := 'True'} : "UDT_DOadv";
      DO11 { S7_SetPoint := 'True'} : "UDT_DOadv";
      DO12 { S7_SetPoint := 'True'} : "UDT_DOadv";
      DO13 { S7_SetPoint := 'True'} : "UDT_DOadv";
      DO14 { S7_SetPoint := 'True'} : "UDT_DOadv";
      DO15 { S7_SetPoint := 'True'} : "UDT_DOadv";
      DO16 { S7_SetPoint := 'True'} : "UDT_DOadv";
   END_VAR
BEGIN
   DO1.iFuncSystemID := 10;
   DO1.iFuncVar := 10;
   DO2.iFuncSystemID := 10;
   DO2.iFuncVar := 11;
   DO3.iFuncSystemID := 10;
   DO3.iFuncVar := 12;
   DO4.iFuncSystemID := 100;
   DO4.iFuncVar := 1;
   DO5.iFuncSystemID := 100;
   DO5.iFuncVar := 5;
   DO6.iFuncSystemID := 100;
   DO6.iFuncVar := 3;
   DO7.iFuncSystemID := 10;
   DO7.iFuncVar := 5;
   DO8.iFuncSystemID := 10;
   DO8.iFuncVar := 6;
   DO9.iFuncSystemID := 10;
   DO9.iFuncVar := 13;
   DO14.iFuncSystemID := 1;
   DO14.iFuncVar := 1;
   DO14.cMOA := 1;
   DO15.iFuncSystemID := 1;
   DO16.iFuncSystemID := 1;
   DO16.iFuncVar := 3;
END_DATA_BLOCK

DATA_BLOCK "SS1_A8_16DI_16DO_DI_Vars"   // DB11081
{ S7_Optimized_Access := 'FALSE' }
VERSION : 0.1
// stored: AutoNumber false, DBAccessibleFromOPCUA true, IsOnlyStoredInLoadMemory false, IsWriteProtectedInAS false
   VAR
      DI1 : "UDT_DIadv";
      DI2 : "UDT_DIadv";
      DI3 : "UDT_DIadv";
      DI4 : "UDT_DIadv";
      DI5 : "UDT_DIadv";
      DI6 : "UDT_DIadv";
      DI7 : "UDT_DIadv";
      DI8 : "UDT_DIadv";
      DI9 { S7_SetPoint := 'True'} : "UDT_DIadv";
      DI10 { S7_SetPoint := 'True'} : "UDT_DIadv";
      DI11 { S7_SetPoint := 'True'} : "UDT_DIadv";
      DI12 { S7_SetPoint := 'True'} : "UDT_DIadv";
      DI13 { S7_SetPoint := 'True'} : "UDT_DIadv";
      DI14 { S7_SetPoint := 'True'} : "UDT_DIadv";
      DI15 { S7_SetPoint := 'True'} : "UDT_DIadv";
      DI16 { S7_SetPoint := 'True'} : "UDT_DIadv";
   END_VAR
BEGIN
   DI1.cFuncSystemID := 1;
   DI1.cFuncVar := 11;
   DI2.cFuncSystemID := 1;
   DI3.cFuncSystemID := 1;
   DI4.cFuncSystemID := 1;
   DI4.cFuncVar := 6;
   DI5.cFuncSystemID := 1;
   DI5.cFuncVar := 4;
   DI6.cFuncSystemID := 1;
   DI6.cFuncVar := 21;
   DI7.cFuncSystemID := 1;
   DI8.cFuncSystemID := 1;
   DI9.cFuncSystemID := 1;
   DI10.cFuncSystemID := 3;
   DI10.cFuncVar := 13;
   DI11.cFuncSystemID := 3;
   DI12.cFuncSystemID := 3;
   DI13.cFuncSystemID := 3;
   DI13.cFuncVar := 3;
   DI14.cFuncSystemID := 3;
   DI14.cFuncVar := 3;
   DI15.cFuncSystemID := 3;
   DI15.cFuncVar := 14;
   DI16.cFuncSystemID := 3;
END_DATA_BLOCK

DATA_BLOCK "SS1_A8_16DI_16DO_DO_Vars"   // DB11082
{ S7_Optimized_Access := 'FALSE' }
VERSION : 0.1
// stored: AutoNumber false, DBAccessibleFromOPCUA true, IsOnlyStoredInLoadMemory false, IsWriteProtectedInAS false
   VAR
      DO1 { S7_SetPoint := 'True'} : "UDT_DOadv";
      DO2 { S7_SetPoint := 'True'} : "UDT_DOadv";
      DO3 { S7_SetPoint := 'True'} : "UDT_DOadv";
      DO4 { S7_SetPoint := 'True'} : "UDT_DOadv";
      DO5 { S7_SetPoint := 'True'} : "UDT_DOadv";
      DO6 { S7_SetPoint := 'True'} : "UDT_DOadv";
      DO7 { S7_SetPoint := 'True'} : "UDT_DOadv";
      DO8 { S7_SetPoint := 'True'} : "UDT_DOadv";
      DO9 { S7_SetPoint := 'True'} : "UDT_DOadv";
      DO10 { S7_SetPoint := 'True'} : "UDT_DOadv";
      DO11 { S7_SetPoint := 'True'} : "UDT_DOadv";
      DO12 { S7_SetPoint := 'True'} : "UDT_DOadv";
      DO13 { S7_SetPoint := 'True'} : "UDT_DOadv";
      DO14 { S7_SetPoint := 'True'} : "UDT_DOadv";
      DO15 { S7_SetPoint := 'True'} : "UDT_DOadv";
      DO16 { S7_SetPoint := 'True'} : "UDT_DOadv";
   END_VAR
BEGIN
   DO1.iFuncSystemID := 1;
   DO1.iFuncVar := 4;
   DO2.iFuncSystemID := 1;
   DO3.iFuncSystemID := 1;
   DO4.iFuncSystemID := 1;
   DO5.iFuncSystemID := 1;
   DO6.cMOA := 1;
   DO7.iFuncSystemID := 3;
   DO7.iFuncVar := 1;
   DO7.cMOA := 1;
   DO8.iFuncSystemID := 3;
   DO9.iFuncSystemID := 3;
   DO9.iFuncVar := 3;
   DO13.iFuncSystemID := 10;
   DO13.iFuncVar := 1;
   DO14.iFuncSystemID := 10;
   DO14.iFuncVar := 2;
   DO15.iFuncSystemID := 10;
   DO15.iFuncVar := 3;
   DO16.iFuncSystemID := 10;
   DO16.iFuncVar := 4;
END_DATA_BLOCK

DATA_BLOCK "SS2_A1_8RTD_AI_Vars"   // DB11121
{ S7_Optimized_Access := 'FALSE' }
VERSION : 0.1
// stored: AutoNumber false, DBAccessibleFromOPCUA true, IsOnlyStoredInLoadMemory false, IsWriteProtectedInAS false
   VAR
      AI1 { S7_SetPoint := 'True'} : "UDT_RTDadv";
      AI2 { S7_SetPoint := 'True'} : "UDT_RTDadv";
      AI3 { S7_SetPoint := 'True'} : "UDT_RTDadv";
      AI4 { S7_SetPoint := 'True'} : "UDT_RTDadv";
      AI5 { S7_SetPoint := 'True'} : "UDT_RTDadv";
      AI6 { S7_SetPoint := 'True'} : "UDT_RTDadv";
      AI7 { S7_SetPoint := 'True'} : "UDT_RTDadv";
      AI8 { S7_SetPoint := 'True'} : "UDT_RTDadv";
   END_VAR
BEGIN
   AI1.cFuncSystemID := 2;
   AI1.cFuncVar := 6;
   AI2.cFuncSystemID := 2;
   AI2.cFuncVar := 4;
   AI3.cFuncSystemID := 2;
   AI3.cFuncVar := 3;
   AI4.cFuncSystemID := 10;
   AI4.cFuncVar := 3;
   AI5.cFuncSystemID := 10;
   AI5.cFuncVar := 5;
   AI6.cFuncSystemID := 10;
   AI6.cFuncVar := 6;
   AI7.cFuncSystemID := 10;
   AI7.cFuncVar := 8;
   AI8.cFuncSystemID := 10;
   AI8.cFuncVar := 9;
END_DATA_BLOCK

DATA_BLOCK "SS2_A3_32DI_DI_Vars"   // DB11141
{ S7_Optimized_Access := 'FALSE' }
VERSION : 0.1
// stored: AutoNumber false, DBAccessibleFromOPCUA true, IsOnlyStoredInLoadMemory false, IsWriteProtectedInAS false
   VAR
      DI1 : "UDT_DIadv";
      DI2 : "UDT_DIadv";
      DI3 : "UDT_DIadv";
      DI4 : "UDT_DIadv";
      DI5 : "UDT_DIadv";
      DI6 : "UDT_DIadv";
      DI7 : "UDT_DIadv";
      DI8 : "UDT_DIadv";
      DI9 { S7_SetPoint := 'True'} : "UDT_DIadv";
      DI10 { S7_SetPoint := 'True'} : "UDT_DIadv";
      DI11 { S7_SetPoint := 'True'} : "UDT_DIadv";
      DI12 { S7_SetPoint := 'True'} : "UDT_DIadv";
      DI13 { S7_SetPoint := 'True'} : "UDT_DIadv";
      DI14 { S7_SetPoint := 'True'} : "UDT_DIadv";
      DI15 { S7_SetPoint := 'True'} : "UDT_DIadv";
      DI16 { S7_SetPoint := 'True'} : "UDT_DIadv";
      DI17 { S7_SetPoint := 'True'} : "UDT_DIadv";
      DI18 { S7_SetPoint := 'True'} : "UDT_DIadv";
      DI19 { S7_SetPoint := 'True'} : "UDT_DIadv";
      DI20 { S7_SetPoint := 'True'} : "UDT_DIadv";
      DI21 { S7_SetPoint := 'True'} : "UDT_DIadv";
      DI22 { S7_SetPoint := 'True'} : "UDT_DIadv";
      DI23 { S7_SetPoint := 'True'} : "UDT_DIadv";
      DI24 { S7_SetPoint := 'True'} : "UDT_DIadv";
      DI25 { S7_SetPoint := 'True'} : "UDT_DIadv";
      DI26 { S7_SetPoint := 'True'} : "UDT_DIadv";
      DI27 { S7_SetPoint := 'True'} : "UDT_DIadv";
      DI28 { S7_SetPoint := 'True'} : "UDT_DIadv";
      DI29 { S7_SetPoint := 'True'} : "UDT_DIadv";
      DI30 { S7_SetPoint := 'True'} : "UDT_DIadv";
      DI31 { S7_SetPoint := 'True'} : "UDT_DIadv";
      DI32 { S7_SetPoint := 'True'} : "UDT_DIadv";
   END_VAR
BEGIN
   DI3.cFuncSystemID := 2;
   DI3.cFuncVar := 0;
   DI4.cFuncSystemID := 2;
   DI4.cFuncVar := 3;
   DI5.cFuncSystemID := 2;
   DI5.cFuncVar := 2;
   DI6.cFuncSystemID := 2;
   DI7.cFuncSystemID := 2;
   DI7.cFuncVar := 14;
   DI8.cFuncSystemID := 2;
   DI9.cFuncSystemID := 2;
   DI9.cFuncVar := 9;
   DI10.cFuncSystemID := 2;
   DI11.cFuncSystemID := 2;
   DI12.cFuncSystemID := 2;
   DI12.cFuncVar := 8;
   DI13.cFuncSystemID := 2;
   DI14.cFuncSystemID := 2;
   DI15.cFuncSystemID := 2;
   DI16.cFuncSystemID := 2;
   DI17.cFuncSystemID := 10;
   DI17.cFuncVar := 35;
   DI18.cFuncSystemID := 10;
   DI18.cFuncVar := 36;
   DI19.cFuncSystemID := 10;
   DI19.cFuncVar := 37;
   DI20.xInversion := true;
   DI20.cFuncSystemID := 10;
   DI20.cFuncVar := 10;
   DI21.xInversion := true;
   DI21.cFuncSystemID := 10;
   DI21.cFuncVar := 13;
   DI22.cFuncSystemID := 10;
   DI22.cFuncVar := 9;
   DI23.cFuncSystemID := 10;
   DI23.cFuncVar := 12;
   DI24.xInversion := true;
   DI24.cFuncSystemID := 10;
   DI24.cFuncVar := 33;
   DI25.cFuncSystemID := 10;
   DI25.cFuncVar := 32;
   DI26.cFuncSystemID := 10;
   DI26.cFuncVar := 14;
   DI27.cFuncSystemID := 10;
   DI27.cFuncVar := 34;
   DI29.cFuncSystemID := 10;
   DI30.cFuncSystemID := 10;
   DI30.cFuncVar := 46;
   DI31.cFuncSystemID := 10;
   DI31.cFuncVar := 44;
END_DATA_BLOCK

DATA_BLOCK "SS2_A2_8AO_AO_Vars"   // DB11131
{ S7_Optimized_Access := 'FALSE' }
VERSION : 0.1
// stored: AutoNumber false, DBAccessibleFromOPCUA true, IsOnlyStoredInLoadMemory false, IsWriteProtectedInAS false
   VAR
      AO1 { S7_SetPoint := 'True'} : "UDT_AOadv";
      AO2 { S7_SetPoint := 'True'} : "UDT_AOadv";
      AO3 : "UDT_AOadv";
      AO4 : "UDT_AOadv";
      AO5 { S7_SetPoint := 'True'} : "UDT_AOadv";
      AO6 { S7_SetPoint := 'True'} : "UDT_AOadv";
      AO7 { S7_SetPoint := 'True'} : "UDT_AOadv";
      AO8 { S7_SetPoint := 'True'} : "UDT_AOadv";
   END_VAR
BEGIN
   AO1.cMOA := 1;
   AO1.cFuncSystemID := 2;
   AO1.cFuncVar := 2;
   AO1.rManOutput := 100.0;
   AO2.cFuncSystemID := 2;
   AO2.cFuncVar := 3;
END_DATA_BLOCK

DATA_BLOCK "SS2_A4_32DO_DO_Vars"   // DB11151
{ S7_Optimized_Access := 'FALSE' }
VERSION : 0.1
// stored: AutoNumber false, DBAccessibleFromOPCUA true, IsOnlyStoredInLoadMemory false, IsWriteProtectedInAS false
   VAR
      DO1 { S7_SetPoint := 'True'} : "UDT_DOadv";
      DO2 { S7_SetPoint := 'True'} : "UDT_DOadv";
      DO3 { S7_SetPoint := 'True'} : "UDT_DOadv";
      DO4 : "UDT_DOadv";
      DO5 { S7_SetPoint := 'True'} : "UDT_DOadv";
      DO6 { S7_SetPoint := 'True'} : "UDT_DOadv";
      DO7 { S7_SetPoint := 'True'} : "UDT_DOadv";
      DO8 { S7_SetPoint := 'True'} : "UDT_DOadv";
      DO9 { S7_SetPoint := 'True'} : "UDT_DOadv";
      DO10 { S7_SetPoint := 'True'} : "UDT_DOadv";
      DO11 { S7_SetPoint := 'True'} : "UDT_DOadv";
      DO12 { S7_SetPoint := 'True'} : "UDT_DOadv";
      DO13 { S7_SetPoint := 'True'} : "UDT_DOadv";
      DO14 { S7_SetPoint := 'True'} : "UDT_DOadv";
      DO15 { S7_SetPoint := 'True'} : "UDT_DOadv";
      DO16 { S7_SetPoint := 'True'} : "UDT_DOadv";
      DO17 { S7_SetPoint := 'True'} : "UDT_DOadv";
      DO18 { S7_SetPoint := 'True'} : "UDT_DOadv";
      DO19 { S7_SetPoint := 'True'} : "UDT_DOadv";
      DO20 { S7_SetPoint := 'True'} : "UDT_DOadv";
      DO21 { S7_SetPoint := 'True'} : "UDT_DOadv";
      DO22 { S7_SetPoint := 'True'} : "UDT_DOadv";
      DO23 { S7_SetPoint := 'True'} : "UDT_DOadv";
      DO24 { S7_SetPoint := 'True'} : "UDT_DOadv";
      DO25 { S7_SetPoint := 'True'} : "UDT_DOadv";
      DO26 { S7_SetPoint := 'True'} : "UDT_DOadv";
      DO27 { S7_SetPoint := 'True'} : "UDT_DOadv";
      DO28 { S7_SetPoint := 'True'} : "UDT_DOadv";
      DO29 { S7_SetPoint := 'True'} : "UDT_DOadv";
      DO30 { S7_SetPoint := 'True'} : "UDT_DOadv";
      DO31 { S7_SetPoint := 'True'} : "UDT_DOadv";
      DO32 { S7_SetPoint := 'True'} : "UDT_DOadv";
   END_VAR
BEGIN
   DO2.iFuncSystemID := 2;
   DO2.iFuncVar := 1;
   DO3.iFuncSystemID := 2;
   DO4.iFuncSystemID := 2;
   DO4.iFuncVar := 3;
   DO5.iFuncSystemID := 10;
   DO5.iFuncVar := 17;
   DO6.iFuncSystemID := 10;
   DO6.iFuncVar := 18;
   DO7.iFuncSystemID := 10;
   DO7.iFuncVar := 7;
   DO8.iFuncSystemID := 10;
   DO8.iFuncVar := 8;
   DO9.iFuncSystemID := 10;
   DO9.iFuncVar := 19;
   DO13.iFuncSystemID := 10;
   DO13.iFuncVar := 16;
END_DATA_BLOCK

DATA_BLOCK "SS2_A5_16DI_DI_Vars"   // DB11161
{ S7_Optimized_Access := 'FALSE' }
VERSION : 0.1
// stored: AutoNumber false, DBAccessibleFromOPCUA true, IsOnlyStoredInLoadMemory false, IsWriteProtectedInAS false
   VAR
      DI1 : "UDT_DIadv";
      DI2 : "UDT_DIadv";
      DI3 : "UDT_DIadv";
      DI4 : "UDT_DIadv";
      DI5 : "UDT_DIadv";
      DI6 : "UDT_DIadv";
      DI7 : "UDT_DIadv";
      DI8 : "UDT_DIadv";
      DI9 { S7_SetPoint := 'True'} : "UDT_DIadv";
      DI10 { S7_SetPoint := 'True'} : "UDT_DIadv";
      DI11 { S7_SetPoint := 'True'} : "UDT_DIadv";
      DI12 { S7_SetPoint := 'True'} : "UDT_DIadv";
      DI13 { S7_SetPoint := 'True'} : "UDT_DIadv";
      DI14 { S7_SetPoint := 'True'} : "UDT_DIadv";
      DI15 { S7_SetPoint := 'True'} : "UDT_DIadv";
      DI16 { S7_SetPoint := 'True'} : "UDT_DIadv";
   END_VAR
BEGIN
   DI1.cFuncSystemID := 2;
   DI1.cFuncVar := 18;
   DI2.cFuncSystemID := 2;
   DI2.cFuncVar := 16;
END_DATA_BLOCK

ORGANIZATION_BLOCK "Main"   // OB1, LAD, ProgramCycle
TITLE = "Main Program Sweep (Cycle)"
{ S7_Optimized_Access := 'TRUE' }
VERSION : 0.1
// stored: AutoNumber true, IsIECCheckEnabled false, SetENOAutomatically false
   VAR_INPUT
      Initial_Call : Bool;   // Initial call of this OB
      Remanence : Bool;   // =True, if remanent data are available
   END_VAR
BEGIN

REGION Network 1: Вже вiдпрацьовано?
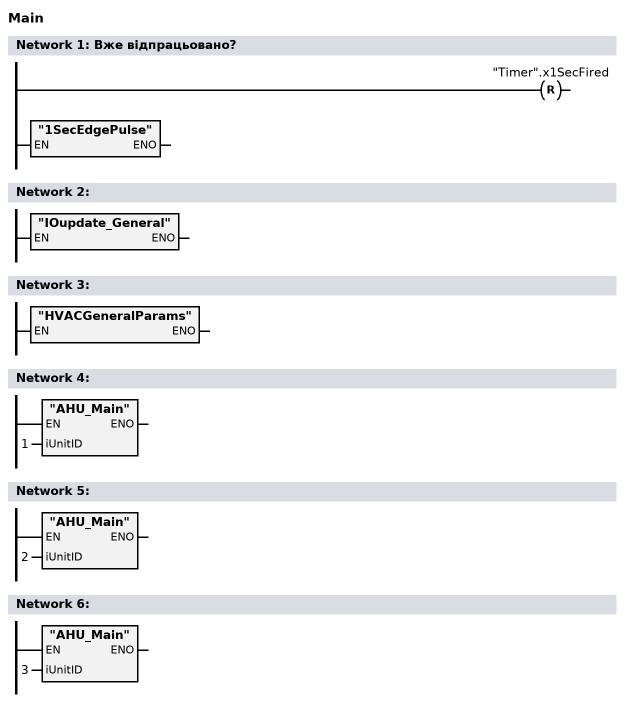
   RUNG wire#powerrail
      R_Coil( "Timer".x1SecFired )
   END_RUNG
   RUNG wire#powerrail
      "1SecEdgePulse"()
   END_RUNG
   // the same network as SCL:
   "Timer".x1SecFired := FALSE;
   "1SecEdgePulse"();
END_REGION

REGION Network 2
   RUNG wire#powerrail
      "IOupdate_General"()
   END_RUNG
   // the same network as SCL:
   "IOupdate_General"();
END_REGION

REGION Network 3
   RUNG wire#powerrail
      "HVACGeneralParams"()
   END_RUNG
   // the same network as SCL:
   "HVACGeneralParams"();
END_REGION

REGION Network 4
   RUNG wire#powerrail
      "AHU_Main"(iUnitID := 1)
   END_RUNG
   // the same network as SCL:
   "AHU_Main"(iUnitID := 1);
END_REGION

REGION Network 5
   RUNG wire#powerrail
      "AHU_Main"(iUnitID := 2)
   END_RUNG
   // the same network as SCL:
   "AHU_Main"(iUnitID := 2);
END_REGION

REGION Network 6
   RUNG wire#powerrail
      "AHU_Main"(iUnitID := 3)
   END_RUNG
   // the same network as SCL:
   "AHU_Main"(iUnitID := 3);
END_REGION

REGION Network 10 (SCL)
   //CASE "Calculated_VariablesF".ModeFromPanel OF
   //    0:  // OFF
   //        "AO_1".FanModulation := 0.0 ;
   //    2:  // Speed1
   //        "AO_1".FanModulation := "Seted_VariablesF".SAFSpeed1;
   //    3:  // Speed2     
   //        "AO_1".FanModulation := "Seted_VariablesF".SAFSpeed2;
   //    ELSE  // Auto
   //        "AO_1".FanModulation := "Seted_VariablesF".SAFSpeedAuto;
   //END_CASE;
END_REGION
END_ORGANIZATION_BLOCK

FUNCTION "1SecEdgePulse" : Void   // FC59999, LAD
{ S7_Optimized_Access := 'TRUE' }
VERSION : 0.1
// stored: AutoNumber false, IsIECCheckEnabled false, SetENOAutomatically false, UDAEnableTagReadback false
BEGIN

REGION Network 1: Одноразовий імпуьс 1сек
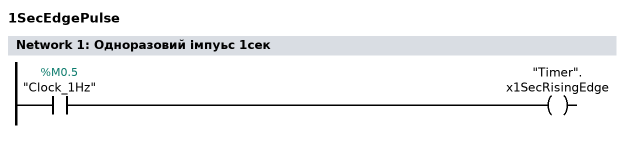
   RUNG wire#powerrail
      Contact( "Clock_1Hz" )
      Coil( "Timer".x1SecRisingEdge )
   END_RUNG
   // the same network as SCL:
   "Timer".x1SecRisingEdge := "Clock_1Hz";
END_REGION

REGION Network 2 (SCL)
   "Timer".x1SecRisingEdge := ("Clock_1Hz" AND NOT "Timer".x1SecPrevClock) AND NOT "Timer".x1SecFired;
   "Timer".x1SecPrevClock := "Clock_1Hz";
   IF "Timer".x1SecRisingEdge THEN
       "Timer".x1SecFired := TRUE;
   END_IF;
END_REGION
END_FUNCTION

FUNCTION "IOupdate_General" : Void   // FC10000, LAD
{ S7_Optimized_Access := 'TRUE' }
VERSION : 0.1
// stored: AutoNumber false, IsIECCheckEnabled false, SetENOAutomatically false, UDAEnableTagReadback false
BEGIN

REGION Network 1
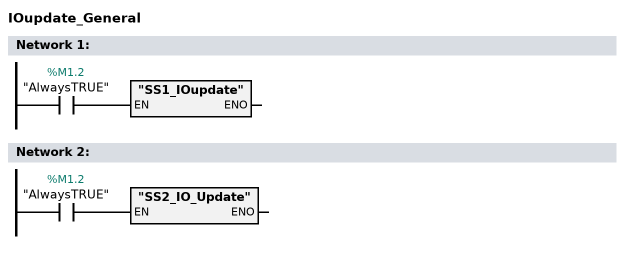
   RUNG wire#powerrail
      Contact( "AlwaysTRUE" )
      "SS1_IOupdate"()
   END_RUNG
   // the same network as SCL:
   IF "AlwaysTRUE" THEN "SS1_IOupdate"(); END_IF;
END_REGION

REGION Network 2
   RUNG wire#powerrail
      Contact( "AlwaysTRUE" )
      "SS2_IO_Update"()
   END_RUNG
   // the same network as SCL:
   IF "AlwaysTRUE" THEN "SS2_IO_Update"(); END_IF;
END_REGION
END_FUNCTION

FUNCTION "SS1_IOupdate" : Void   // FC11000, LAD
{ S7_Optimized_Access := 'TRUE' }
VERSION : 0.1
// stored: AutoNumber false, IsIECCheckEnabled false, SetENOAutomatically false, UDAEnableTagReadback false
BEGIN

REGION Network 1
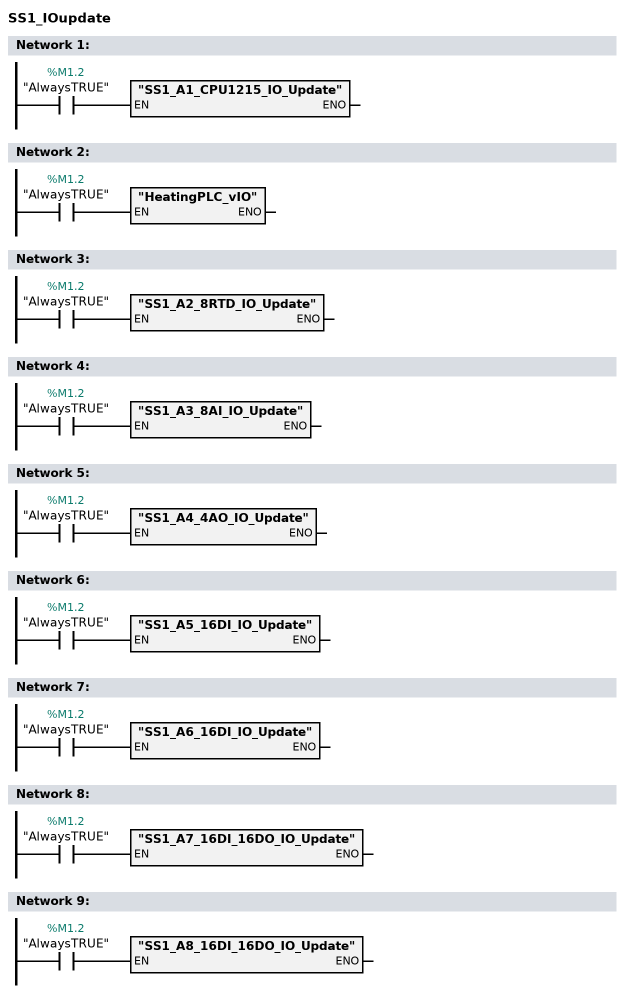
   RUNG wire#powerrail
      Contact( "AlwaysTRUE" )
      "SS1_A1_CPU1215_IO_Update"()
   END_RUNG
   // the same network as SCL:
   IF "AlwaysTRUE" THEN "SS1_A1_CPU1215_IO_Update"(); END_IF;
END_REGION

REGION Network 2
   RUNG wire#powerrail
      Contact( "AlwaysTRUE" )
      "HeatingPLC_vIO"()
   END_RUNG
   // the same network as SCL:
   IF "AlwaysTRUE" THEN "HeatingPLC_vIO"(); END_IF;
END_REGION

REGION Network 3
   RUNG wire#powerrail
      Contact( "AlwaysTRUE" )
      "SS1_A2_8RTD_IO_Update"()
   END_RUNG
   // the same network as SCL:
   IF "AlwaysTRUE" THEN "SS1_A2_8RTD_IO_Update"(); END_IF;
END_REGION

REGION Network 4
   RUNG wire#powerrail
      Contact( "AlwaysTRUE" )
      "SS1_A3_8AI_IO_Update"()
   END_RUNG
   // the same network as SCL:
   IF "AlwaysTRUE" THEN "SS1_A3_8AI_IO_Update"(); END_IF;
END_REGION

REGION Network 5
   RUNG wire#powerrail
      Contact( "AlwaysTRUE" )
      "SS1_A4_4AO_IO_Update"()
   END_RUNG
   // the same network as SCL:
   IF "AlwaysTRUE" THEN "SS1_A4_4AO_IO_Update"(); END_IF;
END_REGION

REGION Network 6
   RUNG wire#powerrail
      Contact( "AlwaysTRUE" )
      "SS1_A5_16DI_IO_Update"()
   END_RUNG
   // the same network as SCL:
   IF "AlwaysTRUE" THEN "SS1_A5_16DI_IO_Update"(); END_IF;
END_REGION

REGION Network 7
   RUNG wire#powerrail
      Contact( "AlwaysTRUE" )
      "SS1_A6_16DI_IO_Update"()
   END_RUNG
   // the same network as SCL:
   IF "AlwaysTRUE" THEN "SS1_A6_16DI_IO_Update"(); END_IF;
END_REGION

REGION Network 8
   RUNG wire#powerrail
      Contact( "AlwaysTRUE" )
      "SS1_A7_16DI_16DO_IO_Update"()
   END_RUNG
   // the same network as SCL:
   IF "AlwaysTRUE" THEN "SS1_A7_16DI_16DO_IO_Update"(); END_IF;
END_REGION

REGION Network 9
   RUNG wire#powerrail
      Contact( "AlwaysTRUE" )
      "SS1_A8_16DI_16DO_IO_Update"()
   END_RUNG
   // the same network as SCL:
   IF "AlwaysTRUE" THEN "SS1_A8_16DI_16DO_IO_Update"(); END_IF;
END_REGION
END_FUNCTION

FUNCTION "SS1_A1_CPU1215_IO_Update" : Void   // FC11010, LAD
{ S7_Optimized_Access := 'TRUE' }
VERSION : 0.1
// stored: AutoNumber false, IsIECCheckEnabled false, SetENOAutomatically false, UDAEnableTagReadback false
BEGIN

REGION Network 1: AI0 / "AI01.1.1" iw64
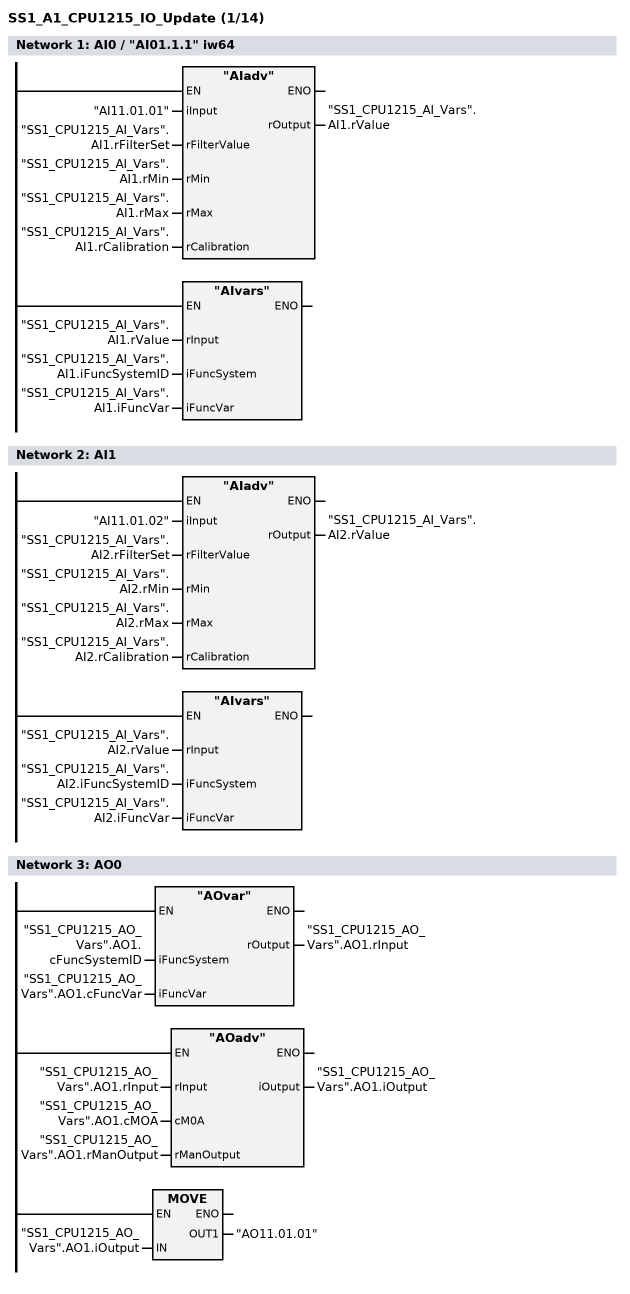
   RUNG wire#powerrail
      "AIadv"(iInput := "AI11.01.01", rFilterValue := "SS1_CPU1215_AI_Vars".AI1.rFilterSet, rMin := "SS1_CPU1215_AI_Vars".AI1.rMin, rMax := "SS1_CPU1215_AI_Vars".AI1.rMax, rCalibration := "SS1_CPU1215_AI_Vars".AI1.rCalibration, rOutput => "SS1_CPU1215_AI_Vars".AI1.rValue)
   END_RUNG
   RUNG wire#powerrail
      "AIvars"(rInput := "SS1_CPU1215_AI_Vars".AI1.rValue, iFuncSystem := "SS1_CPU1215_AI_Vars".AI1.iFuncSystemID, iFuncVar := "SS1_CPU1215_AI_Vars".AI1.iFuncVar)
   END_RUNG
   // the same network as SCL:
   "AIadv"(iInput := "AI11.01.01",
           rFilterValue := "SS1_CPU1215_AI_Vars".AI1.rFilterSet,
           rMin := "SS1_CPU1215_AI_Vars".AI1.rMin,
           rMax := "SS1_CPU1215_AI_Vars".AI1.rMax,
           rCalibration := "SS1_CPU1215_AI_Vars".AI1.rCalibration,
           rOutput => "SS1_CPU1215_AI_Vars".AI1.rValue);
   "AIvars"(rInput := "SS1_CPU1215_AI_Vars".AI1.rValue,
            iFuncSystem := "SS1_CPU1215_AI_Vars".AI1.iFuncSystemID,
            iFuncVar := "SS1_CPU1215_AI_Vars".AI1.iFuncVar);
END_REGION

REGION Network 2: AI1
   RUNG wire#powerrail
      "AIadv"(iInput := "AI11.01.02", rFilterValue := "SS1_CPU1215_AI_Vars".AI2.rFilterSet, rMin := "SS1_CPU1215_AI_Vars".AI2.rMin, rMax := "SS1_CPU1215_AI_Vars".AI2.rMax, rCalibration := "SS1_CPU1215_AI_Vars".AI2.rCalibration, rOutput => "SS1_CPU1215_AI_Vars".AI2.rValue)
   END_RUNG
   RUNG wire#powerrail
      "AIvars"(rInput := "SS1_CPU1215_AI_Vars".AI2.rValue, iFuncSystem := "SS1_CPU1215_AI_Vars".AI2.iFuncSystemID, iFuncVar := "SS1_CPU1215_AI_Vars".AI2.iFuncVar)
   END_RUNG
   // the same network as SCL:
   "AIadv"(iInput := "AI11.01.02",
           rFilterValue := "SS1_CPU1215_AI_Vars".AI2.rFilterSet,
           rMin := "SS1_CPU1215_AI_Vars".AI2.rMin,
           rMax := "SS1_CPU1215_AI_Vars".AI2.rMax,
           rCalibration := "SS1_CPU1215_AI_Vars".AI2.rCalibration,
           rOutput => "SS1_CPU1215_AI_Vars".AI2.rValue);
   "AIvars"(rInput := "SS1_CPU1215_AI_Vars".AI2.rValue,
            iFuncSystem := "SS1_CPU1215_AI_Vars".AI2.iFuncSystemID,
            iFuncVar := "SS1_CPU1215_AI_Vars".AI2.iFuncVar);
END_REGION

REGION Network 3: AO0
   RUNG wire#powerrail
      "AOvar"(iFuncSystem := "SS1_CPU1215_AO_Vars".AO1.cFuncSystemID, iFuncVar := "SS1_CPU1215_AO_Vars".AO1.cFuncVar, rOutput => "SS1_CPU1215_AO_Vars".AO1.rInput)
   END_RUNG
   RUNG wire#powerrail
      "AOadv"(rInput := "SS1_CPU1215_AO_Vars".AO1.rInput, cM0A := "SS1_CPU1215_AO_Vars".AO1.cMOA, rManOutput := "SS1_CPU1215_AO_Vars".AO1.rManOutput, iOutput => "SS1_CPU1215_AO_Vars".AO1.iOutput)
   END_RUNG
   RUNG wire#powerrail
      Move(in := "SS1_CPU1215_AO_Vars".AO1.iOutput, out1 => "AO11.01.01")
   END_RUNG
   // the same network as SCL:
   "AOvar"(iFuncSystem := "SS1_CPU1215_AO_Vars".AO1.cFuncSystemID,
           iFuncVar := "SS1_CPU1215_AO_Vars".AO1.cFuncVar,
           rOutput => "SS1_CPU1215_AO_Vars".AO1.rInput);
   "AOadv"(rInput := "SS1_CPU1215_AO_Vars".AO1.rInput,
           cM0A := "SS1_CPU1215_AO_Vars".AO1.cMOA,
           rManOutput := "SS1_CPU1215_AO_Vars".AO1.rManOutput,
           iOutput => "SS1_CPU1215_AO_Vars".AO1.iOutput);
   "AO11.01.01" := "SS1_CPU1215_AO_Vars".AO1.iOutput;
END_REGION

REGION Network 4: AO1
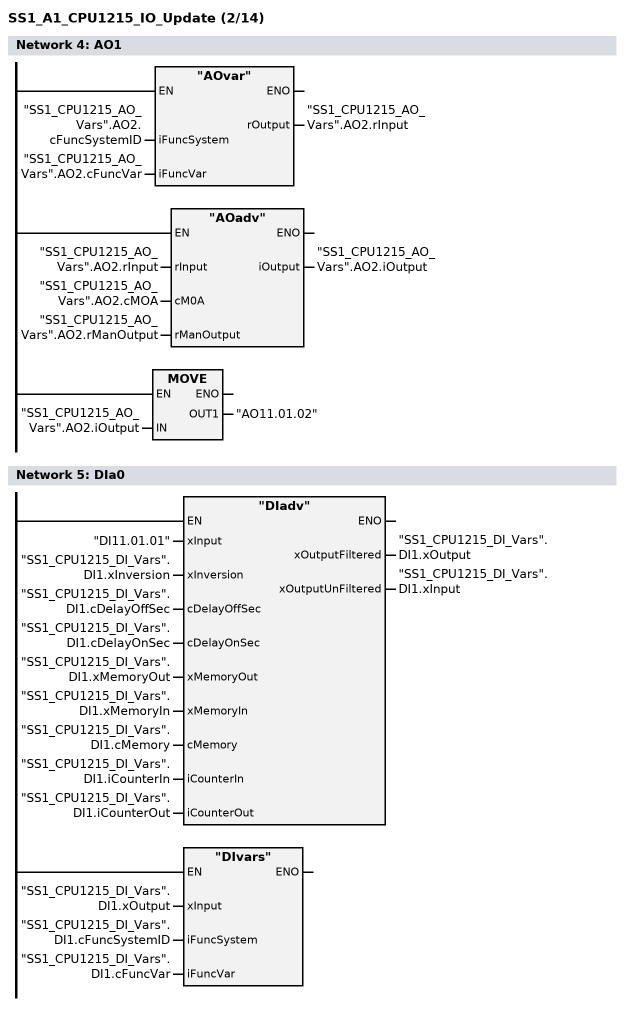
   RUNG wire#powerrail
      "AOvar"(iFuncSystem := "SS1_CPU1215_AO_Vars".AO2.cFuncSystemID, iFuncVar := "SS1_CPU1215_AO_Vars".AO2.cFuncVar, rOutput => "SS1_CPU1215_AO_Vars".AO2.rInput)
   END_RUNG
   RUNG wire#powerrail
      "AOadv"(rInput := "SS1_CPU1215_AO_Vars".AO2.rInput, cM0A := "SS1_CPU1215_AO_Vars".AO2.cMOA, rManOutput := "SS1_CPU1215_AO_Vars".AO2.rManOutput, iOutput => "SS1_CPU1215_AO_Vars".AO2.iOutput)
   END_RUNG
   RUNG wire#powerrail
      Move(in := "SS1_CPU1215_AO_Vars".AO2.iOutput, out1 => "AO11.01.02")
   END_RUNG
   // the same network as SCL:
   "AOvar"(iFuncSystem := "SS1_CPU1215_AO_Vars".AO2.cFuncSystemID,
           iFuncVar := "SS1_CPU1215_AO_Vars".AO2.cFuncVar,
           rOutput => "SS1_CPU1215_AO_Vars".AO2.rInput);
   "AOadv"(rInput := "SS1_CPU1215_AO_Vars".AO2.rInput,
           cM0A := "SS1_CPU1215_AO_Vars".AO2.cMOA,
           rManOutput := "SS1_CPU1215_AO_Vars".AO2.rManOutput,
           iOutput => "SS1_CPU1215_AO_Vars".AO2.iOutput);
   "AO11.01.02" := "SS1_CPU1215_AO_Vars".AO2.iOutput;
END_REGION

REGION Network 5: DIa0
   RUNG wire#powerrail
      "DIadv"(xInput := "DI11.01.01", xInversion := "SS1_CPU1215_DI_Vars".DI1.xInversion, cDelayOffSec := "SS1_CPU1215_DI_Vars".DI1.cDelayOffSec, cDelayOnSec := "SS1_CPU1215_DI_Vars".DI1.cDelayOnSec, xMemoryOut := "SS1_CPU1215_DI_Vars".DI1.xMemoryOut, xMemoryIn := "SS1_CPU1215_DI_Vars".DI1.xMemoryIn, cMemory := "SS1_CPU1215_DI_Vars".DI1.cMemory, xOutputFiltered => "SS1_CPU1215_DI_Vars".DI1.xOutput, xOutputUnFiltered => "SS1_CPU1215_DI_Vars".DI1.xInput, iCounterIn := "SS1_CPU1215_DI_Vars".DI1.iCounterIn, iCounterOut := "SS1_CPU1215_DI_Vars".DI1.iCounterOut)
   END_RUNG
   RUNG wire#powerrail
      "DIvars"(xInput := "SS1_CPU1215_DI_Vars".DI1.xOutput, iFuncSystem := "SS1_CPU1215_DI_Vars".DI1.cFuncSystemID, iFuncVar := "SS1_CPU1215_DI_Vars".DI1.cFuncVar)
   END_RUNG
   // the same network as SCL:
   "DIadv"(xInput := "DI11.01.01",
           xInversion := "SS1_CPU1215_DI_Vars".DI1.xInversion,
           cDelayOffSec := "SS1_CPU1215_DI_Vars".DI1.cDelayOffSec,
           cDelayOnSec := "SS1_CPU1215_DI_Vars".DI1.cDelayOnSec,
           xMemoryOut := "SS1_CPU1215_DI_Vars".DI1.xMemoryOut,
           xMemoryIn := "SS1_CPU1215_DI_Vars".DI1.xMemoryIn,
           cMemory := "SS1_CPU1215_DI_Vars".DI1.cMemory,
           iCounterIn := "SS1_CPU1215_DI_Vars".DI1.iCounterIn,
           iCounterOut := "SS1_CPU1215_DI_Vars".DI1.iCounterOut,
           xOutputFiltered => "SS1_CPU1215_DI_Vars".DI1.xOutput,
           xOutputUnFiltered => "SS1_CPU1215_DI_Vars".DI1.xInput);
   "DIvars"(xInput := "SS1_CPU1215_DI_Vars".DI1.xOutput,
            iFuncSystem := "SS1_CPU1215_DI_Vars".DI1.cFuncSystemID,
            iFuncVar := "SS1_CPU1215_DI_Vars".DI1.cFuncVar);
END_REGION

REGION Network 6: DIa1
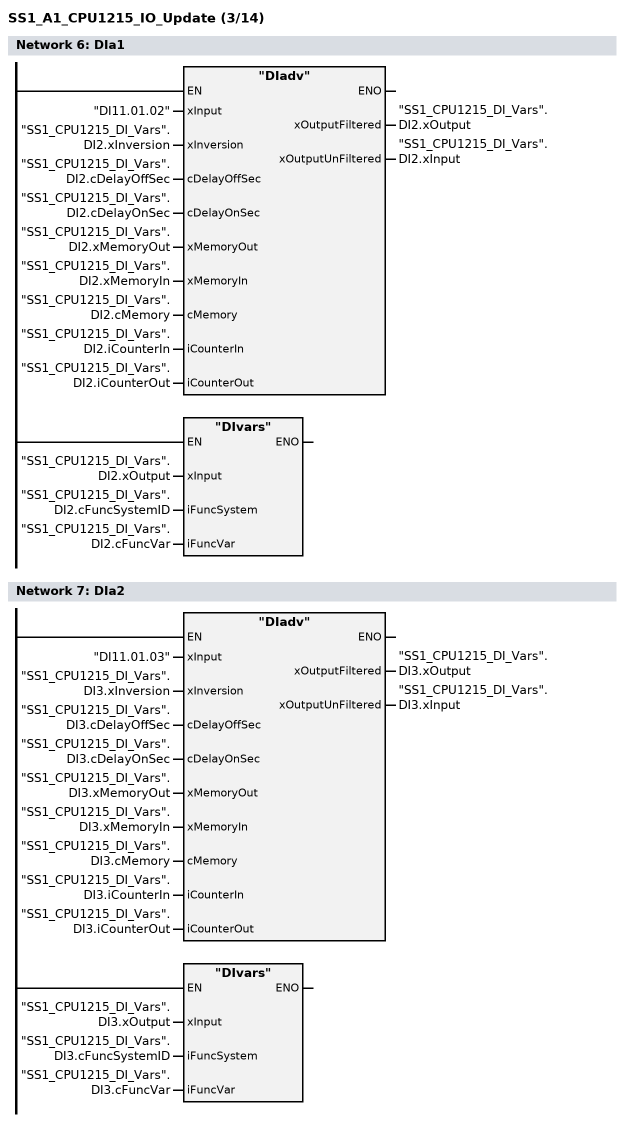
   RUNG wire#powerrail
      "DIadv"(xInput := "DI11.01.02", xInversion := "SS1_CPU1215_DI_Vars".DI2.xInversion, cDelayOffSec := "SS1_CPU1215_DI_Vars".DI2.cDelayOffSec, cDelayOnSec := "SS1_CPU1215_DI_Vars".DI2.cDelayOnSec, xMemoryOut := "SS1_CPU1215_DI_Vars".DI2.xMemoryOut, xMemoryIn := "SS1_CPU1215_DI_Vars".DI2.xMemoryIn, cMemory := "SS1_CPU1215_DI_Vars".DI2.cMemory, xOutputFiltered => "SS1_CPU1215_DI_Vars".DI2.xOutput, xOutputUnFiltered => "SS1_CPU1215_DI_Vars".DI2.xInput, iCounterIn := "SS1_CPU1215_DI_Vars".DI2.iCounterIn, iCounterOut := "SS1_CPU1215_DI_Vars".DI2.iCounterOut)
   END_RUNG
   RUNG wire#powerrail
      "DIvars"(xInput := "SS1_CPU1215_DI_Vars".DI2.xOutput, iFuncSystem := "SS1_CPU1215_DI_Vars".DI2.cFuncSystemID, iFuncVar := "SS1_CPU1215_DI_Vars".DI2.cFuncVar)
   END_RUNG
   // the same network as SCL:
   "DIadv"(xInput := "DI11.01.02",
           xInversion := "SS1_CPU1215_DI_Vars".DI2.xInversion,
           cDelayOffSec := "SS1_CPU1215_DI_Vars".DI2.cDelayOffSec,
           cDelayOnSec := "SS1_CPU1215_DI_Vars".DI2.cDelayOnSec,
           xMemoryOut := "SS1_CPU1215_DI_Vars".DI2.xMemoryOut,
           xMemoryIn := "SS1_CPU1215_DI_Vars".DI2.xMemoryIn,
           cMemory := "SS1_CPU1215_DI_Vars".DI2.cMemory,
           iCounterIn := "SS1_CPU1215_DI_Vars".DI2.iCounterIn,
           iCounterOut := "SS1_CPU1215_DI_Vars".DI2.iCounterOut,
           xOutputFiltered => "SS1_CPU1215_DI_Vars".DI2.xOutput,
           xOutputUnFiltered => "SS1_CPU1215_DI_Vars".DI2.xInput);
   "DIvars"(xInput := "SS1_CPU1215_DI_Vars".DI2.xOutput,
            iFuncSystem := "SS1_CPU1215_DI_Vars".DI2.cFuncSystemID,
            iFuncVar := "SS1_CPU1215_DI_Vars".DI2.cFuncVar);
END_REGION

REGION Network 7: DIa2
   RUNG wire#powerrail
      "DIadv"(xInput := "DI11.01.03", xInversion := "SS1_CPU1215_DI_Vars".DI3.xInversion, cDelayOffSec := "SS1_CPU1215_DI_Vars".DI3.cDelayOffSec, cDelayOnSec := "SS1_CPU1215_DI_Vars".DI3.cDelayOnSec, xMemoryOut := "SS1_CPU1215_DI_Vars".DI3.xMemoryOut, xMemoryIn := "SS1_CPU1215_DI_Vars".DI3.xMemoryIn, cMemory := "SS1_CPU1215_DI_Vars".DI3.cMemory, xOutputFiltered => "SS1_CPU1215_DI_Vars".DI3.xOutput, xOutputUnFiltered => "SS1_CPU1215_DI_Vars".DI3.xInput, iCounterIn := "SS1_CPU1215_DI_Vars".DI3.iCounterIn, iCounterOut := "SS1_CPU1215_DI_Vars".DI3.iCounterOut)
   END_RUNG
   RUNG wire#powerrail
      "DIvars"(xInput := "SS1_CPU1215_DI_Vars".DI3.xOutput, iFuncSystem := "SS1_CPU1215_DI_Vars".DI3.cFuncSystemID, iFuncVar := "SS1_CPU1215_DI_Vars".DI3.cFuncVar)
   END_RUNG
   // the same network as SCL:
   "DIadv"(xInput := "DI11.01.03",
           xInversion := "SS1_CPU1215_DI_Vars".DI3.xInversion,
           cDelayOffSec := "SS1_CPU1215_DI_Vars".DI3.cDelayOffSec,
           cDelayOnSec := "SS1_CPU1215_DI_Vars".DI3.cDelayOnSec,
           xMemoryOut := "SS1_CPU1215_DI_Vars".DI3.xMemoryOut,
           xMemoryIn := "SS1_CPU1215_DI_Vars".DI3.xMemoryIn,
           cMemory := "SS1_CPU1215_DI_Vars".DI3.cMemory,
           iCounterIn := "SS1_CPU1215_DI_Vars".DI3.iCounterIn,
           iCounterOut := "SS1_CPU1215_DI_Vars".DI3.iCounterOut,
           xOutputFiltered => "SS1_CPU1215_DI_Vars".DI3.xOutput,
           xOutputUnFiltered => "SS1_CPU1215_DI_Vars".DI3.xInput);
   "DIvars"(xInput := "SS1_CPU1215_DI_Vars".DI3.xOutput,
            iFuncSystem := "SS1_CPU1215_DI_Vars".DI3.cFuncSystemID,
            iFuncVar := "SS1_CPU1215_DI_Vars".DI3.cFuncVar);
END_REGION

REGION Network 8: DIa3
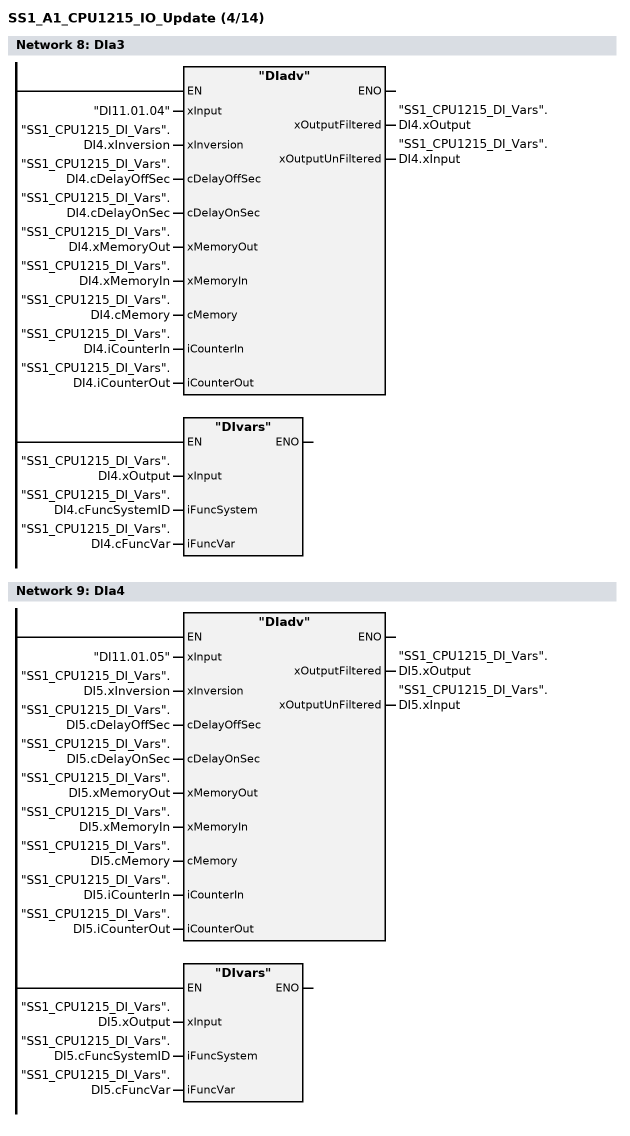
   RUNG wire#powerrail
      "DIadv"(xInput := "DI11.01.04", xInversion := "SS1_CPU1215_DI_Vars".DI4.xInversion, cDelayOffSec := "SS1_CPU1215_DI_Vars".DI4.cDelayOffSec, cDelayOnSec := "SS1_CPU1215_DI_Vars".DI4.cDelayOnSec, xMemoryOut := "SS1_CPU1215_DI_Vars".DI4.xMemoryOut, xMemoryIn := "SS1_CPU1215_DI_Vars".DI4.xMemoryIn, cMemory := "SS1_CPU1215_DI_Vars".DI4.cMemory, xOutputFiltered => "SS1_CPU1215_DI_Vars".DI4.xOutput, xOutputUnFiltered => "SS1_CPU1215_DI_Vars".DI4.xInput, iCounterIn := "SS1_CPU1215_DI_Vars".DI4.iCounterIn, iCounterOut := "SS1_CPU1215_DI_Vars".DI4.iCounterOut)
   END_RUNG
   RUNG wire#powerrail
      "DIvars"(xInput := "SS1_CPU1215_DI_Vars".DI4.xOutput, iFuncSystem := "SS1_CPU1215_DI_Vars".DI4.cFuncSystemID, iFuncVar := "SS1_CPU1215_DI_Vars".DI4.cFuncVar)
   END_RUNG
   // the same network as SCL:
   "DIadv"(xInput := "DI11.01.04",
           xInversion := "SS1_CPU1215_DI_Vars".DI4.xInversion,
           cDelayOffSec := "SS1_CPU1215_DI_Vars".DI4.cDelayOffSec,
           cDelayOnSec := "SS1_CPU1215_DI_Vars".DI4.cDelayOnSec,
           xMemoryOut := "SS1_CPU1215_DI_Vars".DI4.xMemoryOut,
           xMemoryIn := "SS1_CPU1215_DI_Vars".DI4.xMemoryIn,
           cMemory := "SS1_CPU1215_DI_Vars".DI4.cMemory,
           iCounterIn := "SS1_CPU1215_DI_Vars".DI4.iCounterIn,
           iCounterOut := "SS1_CPU1215_DI_Vars".DI4.iCounterOut,
           xOutputFiltered => "SS1_CPU1215_DI_Vars".DI4.xOutput,
           xOutputUnFiltered => "SS1_CPU1215_DI_Vars".DI4.xInput);
   "DIvars"(xInput := "SS1_CPU1215_DI_Vars".DI4.xOutput,
            iFuncSystem := "SS1_CPU1215_DI_Vars".DI4.cFuncSystemID,
            iFuncVar := "SS1_CPU1215_DI_Vars".DI4.cFuncVar);
END_REGION

REGION Network 9: DIa4
   RUNG wire#powerrail
      "DIadv"(xInput := "DI11.01.05", xInversion := "SS1_CPU1215_DI_Vars".DI5.xInversion, cDelayOffSec := "SS1_CPU1215_DI_Vars".DI5.cDelayOffSec, cDelayOnSec := "SS1_CPU1215_DI_Vars".DI5.cDelayOnSec, xMemoryOut := "SS1_CPU1215_DI_Vars".DI5.xMemoryOut, xMemoryIn := "SS1_CPU1215_DI_Vars".DI5.xMemoryIn, cMemory := "SS1_CPU1215_DI_Vars".DI5.cMemory, xOutputFiltered => "SS1_CPU1215_DI_Vars".DI5.xOutput, xOutputUnFiltered => "SS1_CPU1215_DI_Vars".DI5.xInput, iCounterIn := "SS1_CPU1215_DI_Vars".DI5.iCounterIn, iCounterOut := "SS1_CPU1215_DI_Vars".DI5.iCounterOut)
   END_RUNG
   RUNG wire#powerrail
      "DIvars"(xInput := "SS1_CPU1215_DI_Vars".DI5.xOutput, iFuncSystem := "SS1_CPU1215_DI_Vars".DI5.cFuncSystemID, iFuncVar := "SS1_CPU1215_DI_Vars".DI5.cFuncVar)
   END_RUNG
   // the same network as SCL:
   "DIadv"(xInput := "DI11.01.05",
           xInversion := "SS1_CPU1215_DI_Vars".DI5.xInversion,
           cDelayOffSec := "SS1_CPU1215_DI_Vars".DI5.cDelayOffSec,
           cDelayOnSec := "SS1_CPU1215_DI_Vars".DI5.cDelayOnSec,
           xMemoryOut := "SS1_CPU1215_DI_Vars".DI5.xMemoryOut,
           xMemoryIn := "SS1_CPU1215_DI_Vars".DI5.xMemoryIn,
           cMemory := "SS1_CPU1215_DI_Vars".DI5.cMemory,
           iCounterIn := "SS1_CPU1215_DI_Vars".DI5.iCounterIn,
           iCounterOut := "SS1_CPU1215_DI_Vars".DI5.iCounterOut,
           xOutputFiltered => "SS1_CPU1215_DI_Vars".DI5.xOutput,
           xOutputUnFiltered => "SS1_CPU1215_DI_Vars".DI5.xInput);
   "DIvars"(xInput := "SS1_CPU1215_DI_Vars".DI5.xOutput,
            iFuncSystem := "SS1_CPU1215_DI_Vars".DI5.cFuncSystemID,
            iFuncVar := "SS1_CPU1215_DI_Vars".DI5.cFuncVar);
END_REGION

